	3: (* === Wait & process MB response *)
		IF NOT MB_Start THEN
			IF MB_MASTER.MB_Error=0 THEN
				CASE VARS[VarCnt].FunCode OF
					1,2,3,4:
						IF VARS[VarCnt].Variable_Size=200 THEN
							COPY_32SWAP16(ADR(MB_Resp.Data), VARS[VarCnt].Variable);
						ELSIF VARS[VarCnt].Variable_Size>1 THEN
							MEMCPY(ADR(MB_Resp.Data), VARS[VarCnt].Variable, 2*VARS[VarCnt].Variable_Size);
						ELSE
							VARS[VarCnt].Variable^:=MB_Resp.Data[0];
						END_IF
				END_CASE
				MB_Lock:=FALSE;
				(* Signal error recovery *)
				IF VARS_Alarm=TRUE AND VarCnt=VarAlarm THEN
					LogEv(EL_Wrn,EO_MODBUS,ID,5,'');
					VARS_Alarm:=FALSE;
				END_IF
				(* Next var *)
				VarCnt:=VarCnt+1;
				VarSta:=2;
			ELSE
				IF VarRetry<3 THEN
					VarRetry:=VarRetry+1;
					MB_Start:=TRUE;
				ELSE
					MB_Lock:=FALSE;
					(* Signal error *)
					IF VARS_Alarm=FALSE THEN
						LogEv(EL_Wrn,EO_MODBUS,ID,3,INT_TO_STRING(MB_MASTER.MB_Error));
						VARS_Alarm:=TRUE;
						VarAlarm:=VarCnt-1;
					END_IF
					(* Next var *)
					VarCnt:=VarCnt+1;
					VarSta:=2;
				END_IF
			END_IF
		END_IF

ELSE
	VarSta:=0;
END_CASE
END_ACTION

(* POU Utils Functions/TONOF, ST *)
FUNCTION_BLOCK TONOF
VAR_INPUT
	IN		: BOOL;
	PT_ON	: TIME; (* time to pass, before OUT is set *)
	PT_OF	: TIME; (* time to pass, before OUT is reset *)
END_VAR
VAR_OUTPUT
	OUT		: BOOL;
END_VAR
VAR
	timer	: TON;
END_VAR
IF IN<>OUT THEN
	timer(IN:=TRUE,PT:=SEL(IN,PT_OF,PT_ON));
	IF timer.Q THEN OUT:=IN; END_IF
ELSE
	timer(IN:=FALSE);
END_IF
END_FUNCTION_BLOCK

(* POU Plant_Objects/obj_COMPRESSORE_OLD, ST *)
FUNCTION_BLOCK obj_COMPRESSORE_OLD
VAR CONSTANT

	TimeOutModBus: TON;

END_VAR
VAR_INPUT
	ID			:	BYTE;
	Address		:	BYTE;


	(* Modbus *)
	Refresh_Now	:	BOOL;			(* Richiesta di lettura stato macchina Immediata  *)
	retryErrMax	:	BYTE := 2;

	OnOff		: 	BOOL;

	IndirizzoDaScrivere: WORD;
	DatoDaScrivere: INT;
	ScriviDato: BOOL;
	ScriviCoil: BOOL;

	fWriteAttivazioneComandi:BOOL;


	RUN_REQ: BOOL;
	STOP_REQ:BOOL;
	AgggiornoStartStop: BOOL;

	CARICO_REQ: BOOL;
	RELEASE_REQ: BOOL;

	LocSelManAuto:BOOL;
	LocOFP:INT;
	LocONP:INT;


END_VAR
VAR_IN_OUT
	ModBus		:obj_MODBUS;
END_VAR
VAR_OUTPUT
	Run			:	BOOL;

	Status_Log	:	WORD;
	Status_Vis	:	DWORD;
END_VAR
VAR
	(* da diego per gestione stato stringa > 255*)
	temp :STRING(255);
	tempRaw		: ARRAY [0..MAX_SEND_TCP_CLIENT] OF BYTE;
	tempRawLen :DINT;
	longString:STRING(255);

	(* Timer manage switch on/off delay *)
	Delay		: 	TONOF;
	Warning		:	FLT_TAP := (TAP:=100);
	AllarmeCompressore_MB		:	FLT_TAP;
	WarningCompressore_MB		:	FLT_TAP;
	AllarmeCompressoreAttivo_MB		:	FLT_TAP;
	RientrAllarmeCompressore_MB		:	FLT_TAP;
	RientrWarningCompressore_MB		:	FLT_TAP;

	AllarmeAttivo: INT;


	state		:	INT;
	retry		:	BYTE;
	retryErr	:	BYTE;
	ReadTmr		:	TON := (PT:=T#5s);
	fModbusAlr:BOOL;

	Ctrl_Run: BOOL;


	VerificaFuctionCode: INT;
	VerificaNodoLetto: INT;
	ErroreComuModBus: BOOL;
	IndiceErrore: BYTE;

	MB_BitStato: ARRAY [0..1] OF BOOL;
	MB_RegistriLetti: ARRAY [0..1] OF INT;
	MB_RegistriHoldingLetti: ARRAY [0..400] OF INT;
	MB_BitStatoCoil: ARRAY [0..1] OF BOOL;



	AddressRead: BYTE;
	index: BYTE;
	indexErr: BYTE;

	x: INT;
	IndirizzoStart: INT;
	Stop: BOOL;
	start: BOOL;
	StatusControl: ARRAY [0..15] OF BOOL;



	TOFF_RitardoAllarme: TOF;
	TOFF_RitardoWarning: TOF;
	trig_RitardoWarning: F_TRIG;
	trig_Ritardoallarme: F_TRIG;
	CompressoreInAllarme: BOOL;
	AllarmeAttivoSuCompressore: INT;
	CompressoreInWarning: BOOL;
	WarningAttivoSuCompressore: INT;
END_VAR
(* Call ModBus state machine *)
Stm();

(* Check alarm	*)
CheckAlarm();

(* Seganalzione stato Compressore  *)
IF ErroreComuModBus OR AllarmeCompressoreAttivo_MB.IN THEN (* corretto da DB 27/07/2017, era AllarmeCompressore_MB*)
		Status_Log:=2; Status_Vis:=16#2020F0;
   ELSIF WarningCompressore_MB.in  THEN
		Status_Log:=1; Status_Vis:=16#20F0F0;
    ELSE
		Status_Log:=0;
		Status_Vis:=16#006000;
END_IF
END_FUNCTION_BLOCK
ACTION AddLogData:
Logger.s1:=INSERT('&COMPINGRML=',BYTE_TO_STRING(ID),11);
IF ID<10 THEN Logger.s1:=INSERT(Logger.s1,'0',11); END_IF

FOR tempRawLen:=0 TO MAX_SEND_TCP_CLIENT DO
                tempRaw[tempRawLen]:=0;
END_FOR

tempRawLen:=0;


temp:=Logger.s1;
ADDSTRING(ADR(tempRaw), ADR(temp), tempRawLen);



temp:=CONCAT(WORD_TO_STRING(Status_Log),';');
ADDSTRING(ADR(tempRaw), ADR(temp), tempRawLen);


(* Sparo gli ingressi Digitali **)
FOR x:= 0 TO 15 DO
	temp:=CONCAT(SEL(StatusControl[x],'0','1'),';');
	ADDSTRING(ADR(tempRaw), ADR(temp), tempRawLen);
END_FOR

(*

temp:=CONCAT(INT_TO_STRING(MB_RegistriHoldingLetti[1]),';');
ADDSTRING(ADR(tempRaw), ADR(temp), tempRawLen);
temp:=CONCAT(INT_TO_STRING(MB_RegistriHoldingLetti[1]),';');
ADDSTRING(ADR(tempRaw), ADR(temp), tempRawLen); *)
temp:=CONCAT(INT_TO_STRING(MB_RegistriHoldingLetti[3]),';');
ADDSTRING(ADR(tempRaw), ADR(temp), tempRawLen);
temp:=CONCAT(INT_TO_STRING(MB_RegistriHoldingLetti[4]),';');
ADDSTRING(ADR(tempRaw), ADR(temp), tempRawLen);
temp:=CONCAT(INT_TO_STRING(MB_RegistriHoldingLetti[5]),';');
ADDSTRING(ADR(tempRaw), ADR(temp), tempRawLen);
temp:=CONCAT(INT_TO_STRING(MB_RegistriHoldingLetti[6]),';');
ADDSTRING(ADR(tempRaw), ADR(temp), tempRawLen);
temp:=CONCAT(INT_TO_STRING(MB_RegistriHoldingLetti[7]),';');
ADDSTRING(ADR(tempRaw), ADR(temp), tempRawLen);
temp:=CONCAT(INT_TO_STRING(MB_RegistriHoldingLetti[8]),';');
ADDSTRING(ADR(tempRaw), ADR(temp), tempRawLen);
temp:=CONCAT(INT_TO_STRING(MB_RegistriHoldingLetti[9]),';');
ADDSTRING(ADR(tempRaw), ADR(temp), tempRawLen);
temp:=CONCAT(INT_TO_STRING(MB_RegistriHoldingLetti[10]),';');
ADDSTRING(ADR(tempRaw), ADR(temp), tempRawLen);
temp:=CONCAT(INT_TO_STRING(MB_RegistriHoldingLetti[20]),';');
ADDSTRING(ADR(tempRaw), ADR(temp), tempRawLen);
temp:=CONCAT(INT_TO_STRING(MB_RegistriHoldingLetti[64]),';');
ADDSTRING(ADR(tempRaw), ADR(temp), tempRawLen);
temp:=CONCAT(INT_TO_STRING(MB_RegistriHoldingLetti[65]),';');
ADDSTRING(ADR(tempRaw), ADR(temp), tempRawLen);
temp:=CONCAT(INT_TO_STRING(MB_RegistriHoldingLetti[66]),';');
ADDSTRING(ADR(tempRaw), ADR(temp), tempRawLen);
temp:=CONCAT(INT_TO_STRING(MB_RegistriHoldingLetti[67]),';');
ADDSTRING(ADR(tempRaw), ADR(temp), tempRawLen);
temp:=CONCAT(INT_TO_STRING(MB_RegistriHoldingLetti[98]),';');
ADDSTRING(ADR(tempRaw), ADR(temp), tempRawLen);
temp:=CONCAT(INT_TO_STRING(MB_RegistriHoldingLetti[103]),';');
ADDSTRING(ADR(tempRaw), ADR(temp), tempRawLen);
temp:=CONCAT(INT_TO_STRING(MB_RegistriHoldingLetti[112]),';');
ADDSTRING(ADR(tempRaw), ADR(temp), tempRawLen);
temp:=CONCAT(INT_TO_STRING(MB_RegistriHoldingLetti[113]),';');
ADDSTRING(ADR(tempRaw), ADR(temp), tempRawLen);
temp:=CONCAT(INT_TO_STRING(MB_RegistriHoldingLetti[114]),';');
ADDSTRING(ADR(tempRaw), ADR(temp), tempRawLen);
temp:=CONCAT(INT_TO_STRING(MB_RegistriHoldingLetti[116]),';');
ADDSTRING(ADR(tempRaw), ADR(temp), tempRawLen);
temp:=CONCAT(INT_TO_STRING(MB_RegistriHoldingLetti[117]),';');
ADDSTRING(ADR(tempRaw), ADR(temp), tempRawLen);
temp:=CONCAT(INT_TO_STRING(MB_RegistriHoldingLetti[123]),';');
ADDSTRING(ADR(tempRaw), ADR(temp), tempRawLen);
temp:=CONCAT(INT_TO_STRING(MB_RegistriHoldingLetti[125]),';');
ADDSTRING(ADR(tempRaw), ADR(temp), tempRawLen);
temp:=CONCAT(INT_TO_STRING(MB_RegistriHoldingLetti[130]),';');
ADDSTRING(ADR(tempRaw), ADR(temp), tempRawLen);
temp:=CONCAT(INT_TO_STRING(MB_RegistriHoldingLetti[255]),';');
ADDSTRING(ADR(tempRaw), ADR(temp), tempRawLen);
temp:=CONCAT(INT_TO_STRING(MB_RegistriHoldingLetti[256]),';');
ADDSTRING(ADR(tempRaw), ADR(temp), tempRawLen);
temp:=CONCAT(INT_TO_STRING(MB_RegistriHoldingLetti[257]),';');
ADDSTRING(ADR(tempRaw), ADR(temp), tempRawLen);
temp:=CONCAT(INT_TO_STRING(MB_RegistriHoldingLetti[258]),';');
ADDSTRING(ADR(tempRaw), ADR(temp), tempRawLen);
temp:=CONCAT(INT_TO_STRING(MB_RegistriHoldingLetti[259]),';');
ADDSTRING(ADR(tempRaw), ADR(temp), tempRawLen);
temp:=CONCAT(INT_TO_STRING(MB_RegistriHoldingLetti[260]),';');
ADDSTRING(ADR(tempRaw), ADR(temp), tempRawLen);
temp:=CONCAT(INT_TO_STRING(MB_RegistriHoldingLetti[261]),';');
ADDSTRING(ADR(tempRaw), ADR(temp), tempRawLen);
temp:=CONCAT(INT_TO_STRING(MB_RegistriHoldingLetti[261]),';');
ADDSTRING(ADR(tempRaw), ADR(temp), tempRawLen);
temp:=CONCAT(INT_TO_STRING(MB_RegistriHoldingLetti[263]),';');
ADDSTRING(ADR(tempRaw), ADR(temp), tempRawLen);
temp:=CONCAT(INT_TO_STRING(MB_RegistriHoldingLetti[264]),';');
ADDSTRING(ADR(tempRaw), ADR(temp), tempRawLen);
temp:=CONCAT(INT_TO_STRING(MB_RegistriHoldingLetti[265]),';');
ADDSTRING(ADR(tempRaw), ADR(temp), tempRawLen);
temp:=CONCAT(INT_TO_STRING(MB_RegistriHoldingLetti[266]),';');
ADDSTRING(ADR(tempRaw), ADR(temp), tempRawLen);
temp:=CONCAT(INT_TO_STRING(MB_RegistriHoldingLetti[267]),';');
ADDSTRING(ADR(tempRaw), ADR(temp), tempRawLen);
temp:=CONCAT(INT_TO_STRING(MB_RegistriHoldingLetti[268]),';');
ADDSTRING(ADR(tempRaw), ADR(temp), tempRawLen);
temp:=CONCAT(INT_TO_STRING(MB_RegistriHoldingLetti[269]),';');
ADDSTRING(ADR(tempRaw), ADR(temp), tempRawLen);
temp:=(INT_TO_STRING(MB_RegistriHoldingLetti[270]));
ADDSTRING(ADR(tempRaw), ADR(temp), tempRawLen);


ADDSTRING(ADR(Logger.TData), ADR(tempRaw), Logger.TLen);
END_ACTION
ACTION CheckAlarm:
(**** GEstione Log ad Evento *****)



	AllarmeCompressoreAttivo_MB(IN:=CompressoreInAllarme AND AllarmeAttivoSuCompressore<>AllarmeAttivo );

	IF  AllarmeCompressoreAttivo_MB.EVH THEN
		LogEv(EL_Alarm,EO_COMPINGRML,ID,1,CONCAT ('AllarmeAttivo_n.', INT_TO_STRING(MB_RegistriHoldingLetti[256])));
		AllarmeAttivo:=MB_RegistriHoldingLetti[256];
	END_IF


	TOFF_RitardoAllarme(in:=CompressoreInAllarme,pt:=t#10s);    (* AllarmeAttivoSuCompressore=0 *)
	RientrAllarmeCompressore_MB(IN:=(TOFF_RitardoAllarme.Q) );

	IF  RientrAllarmeCompressore_MB.EVL  THEN
		LogEv(EL_Log,EO_COMPINGRML,ID,2,CONCAT ('AllarmeRientrato_n.', INT_TO_STRING(MB_RegistriHoldingLetti[256])));
		AllarmeAttivo:=0;
		AllarmeAttivoSuCompressore:=0;
	END_IF



	WarningCompressore_MB(IN:=CompressoreInWarning );

	IF WarningCompressore_MB.EVH THEN
		LogEv(EL_Wrn,EO_COMPINGRML,ID,1,CONCAT ('WarninigAttivo_n.', INT_TO_STRING(MB_RegistriHoldingLetti[255])));
	END_IF

	TOFF_RitardoWarning(in:=CompressoreInWarning,pt:=t#10s);   (* WarningAttivoSuCompressore=0*)
	RientrWarningCompressore_MB(IN:=(TOFF_RitardoWarning.Q) );

	IF RientrWarningCompressore_MB.EVL THEN
		LogEv(EL_Log,EO_COMPINGRML,ID,2,CONCAT ('WarningRientrato_n.', INT_TO_STRING(MB_RegistriHoldingLetti[255])));
	END_IF
END_ACTION
ACTION Stm:
CASE state OF
	0:	(* Refresh time manager *)
		ReadTmr(IN:=NOT ReadTmr.Q);
		(*A tempo interrogo il nodo sempre che non ci sia qualcuno che lo sta interrogando in quel momento *)

		IF (ReadTmr.Q AND NodoDaInterrogareCompressoreVecchio=Address )  AND NOT InibiscoModbusCompressoreVecchio THEN
			state := 10;
			ReadTmr.PT := T#100ms;  (* moreno *)
			Refresh_Now := FALSE;
			InibiscoModbusCompressoreVecchio := TRUE;
		END_IF

	(**** Leggo le Analogiche a Disposzione  ****)

	10:	(* richiedo lettura Holding Registere   *)

		Modbus.MB_Query.SlaveAddress := Address;
		Modbus.MB_Query.FunctionCode := 3;
		IndirizzoStart:=1;
		ModBus.MB_Query.Read_StartAddress :=IndirizzoStart - 1 ;
		ModBus.MB_Query.Read_Quantity := 2;
		ModBus.MB_Start := TRUE;
		state := 20;

	20:	(* Risposta all'interrogazione *)
		IF NOT ModBus.MB_Start   THEN
			VerificaFuctionCode:=ModBus.MB_Resp.FunctionCode;
			VerificaNodoLetto:=ModBus.MB_Resp.SlaveAddress;

			IF ModBus.MB_MASTER.MB_Error<>0 THEN
				state := 300;
			ELSE
				FOR x:=0 TO ModBus.MB_Query.Read_Quantity DO
					IF x+IndirizzoStart=3 THEN
						IF  ModBus.MB_Resp.Data[x]<260 THEN    (* condizione perchè questo registro si sporca con un valore 599 *)
				       		MB_RegistriHoldingLetti[x+IndirizzoStart] := ModBus.MB_Resp.Data[x];   	(* Vedi tabella *)
						ELSE
				       		MB_RegistriHoldingLetti[x+IndirizzoStart] := MB_RegistriHoldingLetti[x+IndirizzoStart];   	(* Vedi tabella *)
						END_IF
					ELSE
				       	MB_RegistriHoldingLetti[x+IndirizzoStart] := ModBus.MB_Resp.Data[x];   	(* Vedi tabella *)
					END_IF
				END_FOR

					StatusControl[0]:= MB_RegistriHoldingLetti[IndirizzoStart].0;   	(* Vedi tabella *)
					StatusControl[1]:= MB_RegistriHoldingLetti[IndirizzoStart].1;   	(* Vedi tabella *)
					StatusControl[2]:= MB_RegistriHoldingLetti[IndirizzoStart].2;   	(* Vedi tabella *)
					StatusControl[3]:= MB_RegistriHoldingLetti[IndirizzoStart].3;   	(* Vedi tabella *)
					StatusControl[4]:= MB_RegistriHoldingLetti[IndirizzoStart].4;   	(* Vedi tabella *)
					StatusControl[5]:= MB_RegistriHoldingLetti[IndirizzoStart].5;   	(* Vedi tabella *)
					StatusControl[6]:= MB_RegistriHoldingLetti[IndirizzoStart].6;   	(* Vedi tabella *)
					StatusControl[7]:= MB_RegistriHoldingLetti[IndirizzoStart].7;   	(* Vedi tabella *)
					StatusControl[8]:= MB_RegistriHoldingLetti[IndirizzoStart].8;   	(* Vedi tabella *)
					StatusControl[9]:= MB_RegistriHoldingLetti[IndirizzoStart].9;   	(* Vedi tabella *)
					StatusControl[10]:= MB_RegistriHoldingLetti[IndirizzoStart].10;   	(* Vedi tabella *)
					StatusControl[11]:= MB_RegistriHoldingLetti[IndirizzoStart].11;   	(* Vedi tabella *)
					StatusControl[12]:= MB_RegistriHoldingLetti[IndirizzoStart].12;   	(* Vedi tabella *)
					StatusControl[13]:= MB_RegistriHoldingLetti[IndirizzoStart].13;   	(* Vedi tabella *)
					StatusControl[14]:= MB_RegistriHoldingLetti[IndirizzoStart].14;   	(* Vedi tabella *)
					StatusControl[15]:= MB_RegistriHoldingLetti[IndirizzoStart].15;   	(* Vedi tabella *)


					CompressoreInAllarme:=StatusControl[6];
					CompressoreInWarning:=StatusControl[7];



				IndirizzoStart:=3;
				ModBus.MB_Query.Read_StartAddress :=IndirizzoStart-1; 	(* richiedo lettura altri Parametri *)
				ModBus.MB_Query.Read_Quantity := 19;
				ModBus.MB_Start := TRUE;

				state := 40;
			END_IF
		END_IF

	30: (* Rispota Altri paramenti *)
		IF NOT ModBus.MB_Start  THEN

			IF ModBus.MB_MASTER.MB_Error<>0 THEN
				state := 300;
			ELSE

				FOR x:=0 TO ModBus.MB_Query.Read_Quantity DO
					MB_RegistriHoldingLetti[x+IndirizzoStart] := ModBus.MB_Resp.Data[x];   	(* Vedi tabella *)
				END_FOR

				IndirizzoStart:=20;
				ModBus.MB_Query.Read_StartAddress :=IndirizzoStart-1; 	(* richiedo lettura altri Parametri *)
				ModBus.MB_Query.Read_Quantity := 1;
				ModBus.MB_Start := TRUE;

				state := 40;
			END_IF
		END_IF

	40: (* Rispota Altri paramenti *)
		IF NOT ModBus.MB_Start  THEN

			IF ModBus.MB_MASTER.MB_Error<>0 THEN
				state := 300;
			ELSE

				FOR x:=0 TO ModBus.MB_Query.Read_Quantity DO
					MB_RegistriHoldingLetti[x+IndirizzoStart] := ModBus.MB_Resp.Data[x];   	(* Vedi tabella *)
				END_FOR

				IndirizzoStart:=64;
				ModBus.MB_Query.Read_StartAddress :=IndirizzoStart-1; 	(* richiedo lettura altri Parametri *)
				ModBus.MB_Query.Read_Quantity := 4;
				ModBus.MB_Start := TRUE;

				state := 45;
			END_IF
		END_IF

	45: (* Rispota Altri paramenti *)
		IF NOT ModBus.MB_Start  THEN

			IF ModBus.MB_MASTER.MB_Error<>0 THEN
				state := 300;
			ELSE
				FOR x:=0 TO ModBus.MB_Query.Read_Quantity DO
					MB_RegistriHoldingLetti[x+IndirizzoStart] := ModBus.MB_Resp.Data[x];   	(* Vedi tabella *)
				END_FOR

				IndirizzoStart:=96;
				ModBus.MB_Query.Read_StartAddress :=IndirizzoStart-1; 	(* richiedo lettura altri Parametri *)
				ModBus.MB_Query.Read_Quantity := 8;
				ModBus.MB_Start := TRUE;

				state := 50;
			END_IF
		END_IF


	50: (* Rispota Altri paramenti *)
		IF NOT ModBus.MB_Start  THEN

			IF ModBus.MB_MASTER.MB_Error<>0 THEN
				state := 300;
			ELSE
				FOR x:=0 TO ModBus.MB_Query.Read_Quantity DO
					MB_RegistriHoldingLetti[x+IndirizzoStart] := ModBus.MB_Resp.Data[x];   	(* Vedi tabella *)
				END_FOR

				IndirizzoStart:=112;
				ModBus.MB_Query.Read_StartAddress :=IndirizzoStart-1; 	(* richiedo lettura altri Parametri *)
				ModBus.MB_Query.Read_Quantity := 10;
				ModBus.MB_Start := TRUE;


				state := 51;
			END_IF
		END_IF


	51: (* Rispota Altri paramenti *)
		IF NOT ModBus.MB_Start  THEN

			IF ModBus.MB_MASTER.MB_Error<>0 THEN
				state := 300;
			ELSE
				FOR x:=0 TO ModBus.MB_Query.Read_Quantity DO
					MB_RegistriHoldingLetti[x+IndirizzoStart] := ModBus.MB_Resp.Data[x];   	(* Vedi tabella *)
				END_FOR

				IndirizzoStart:=256;
				ModBus.MB_Query.Read_StartAddress :=IndirizzoStart-1; 	(* richiedo lettura altri Parametri *)
				ModBus.MB_Query.Read_Quantity := 14;
				ModBus.MB_Start := TRUE;


				state := 55;
			END_IF
		END_IF


	55: (* Rispota Altri paramenti *)
		IF NOT ModBus.MB_Start  THEN

			IF ModBus.MB_MASTER.MB_Error<>0 THEN
				state := 300;
			ELSE
				FOR x:=0 TO ModBus.MB_Query.Read_Quantity DO
					MB_RegistriHoldingLetti[x+IndirizzoStart] := ModBus.MB_Resp.Data[x];   	(* Vedi tabella *)
				END_FOR

				WarningAttivoSuCompressore:=MB_RegistriHoldingLetti[255];
				AllarmeAttivoSuCompressore:=MB_RegistriHoldingLetti[256];


				IndirizzoStart:=122;
				ModBus.MB_Query.Read_StartAddress :=IndirizzoStart-1; 	(* richiedo lettura altri Parametri *)
				ModBus.MB_Query.Read_Quantity := 10;
				ModBus.MB_Start := TRUE;

				state := 56;
			END_IF
		END_IF

	56: (* Rispota Altri paramenti *)
		IF NOT ModBus.MB_Start  THEN

			IF ModBus.MB_MASTER.MB_Error<>0 THEN
				state := 300;
			ELSE
				FOR x:=0 TO ModBus.MB_Query.Read_Quantity DO
					MB_RegistriHoldingLetti[x+IndirizzoStart] := ModBus.MB_Resp.Data[x];   	(* Vedi tabella *)
				END_FOR

				IndirizzoStart:=132;
				ModBus.MB_Query.Read_StartAddress :=IndirizzoStart-1; 	(* richiedo lettura altri Parametri *)
				ModBus.MB_Query.Read_Quantity := 10;
				ModBus.MB_Start := TRUE;

				state := 57;
			END_IF
		END_IF

	57: (* Rispota Altri paramenti *)
		IF NOT ModBus.MB_Start  THEN

			IF ModBus.MB_MASTER.MB_Error<>0 THEN
				state := 300;
			ELSE
				FOR x:=0 TO ModBus.MB_Query.Read_Quantity DO
					MB_RegistriHoldingLetti[x+IndirizzoStart] := ModBus.MB_Resp.Data[x];   	(* Vedi tabella *)
				END_FOR

				IndirizzoStart:=142;
				ModBus.MB_Query.Read_StartAddress :=IndirizzoStart-1; 	(* richiedo lettura altri Parametri *)
				ModBus.MB_Query.Read_Quantity := 10;
				ModBus.MB_Start := TRUE;

				state := 58;
			END_IF
		END_IF

	58: (* Rispota Altri paramenti *)
		IF NOT ModBus.MB_Start  THEN

			IF ModBus.MB_MASTER.MB_Error<>0 THEN
				state := 300;
			ELSE
				FOR x:=0 TO ModBus.MB_Query.Read_Quantity DO
					MB_RegistriHoldingLetti[x+IndirizzoStart] := ModBus.MB_Resp.Data[x];   	(* Vedi tabella *)
				END_FOR

				IndirizzoStart:=250;
				ModBus.MB_Query.Read_StartAddress :=IndirizzoStart-1; 	(* richiedo lettura altri Parametri *)
				ModBus.MB_Query.Read_Quantity := 6;
				ModBus.MB_Start := TRUE;

				state := 60;
			END_IF
		END_IF




	60: (* Rispota Altri paramenti *)
		IF NOT ModBus.MB_Start  THEN

			IF ModBus.MB_MASTER.MB_Error<>0 THEN
				state := 300;
			ELSE
				FOR x:=0 TO ModBus.MB_Query.Read_Quantity DO
					MB_RegistriHoldingLetti[x+IndirizzoStart] := ModBus.MB_Resp.Data[x];   	(* Vedi tabella *)
				END_FOR

				state :=290;
			END_IF
		END_IF


		290:    (* Scrittura il comando di run o stop da remoto*)
		IF NOT ModBus.MB_Start THEN
			IF ModBus.MB_MASTER.MB_Error<>0 THEN (*OR ModBus.MB_MASTER.MB_Error<>0 THEN*)
				state := 300;
			ELSE
				IF AgggiornoStartStop  THEN

					Modbus.MB_Query.FunctionCode := 6;
					Modbus.MB_Query.SlaveAddress := Address;

					IF RUN_REQ THEN
							IndirizzoDaScrivere:=1;
								 DatoDaScrivere:=MB_RegistriHoldingLetti[IndirizzoDaScrivere];
	  							 DatoDaScrivere.0:=TRUE;
  							        DatoDaScrivere.1:=TRUE;
							        DatoDaScrivere.2:=FALSE;
								 RUN_REQ:=FALSE;
					END_IF
					IF STOP_REQ THEN
							IndirizzoDaScrivere:=1;
								 DatoDaScrivere:=MB_RegistriHoldingLetti[IndirizzoDaScrivere];
	  							 DatoDaScrivere.0:=TRUE;
  							        DatoDaScrivere.1:=FALSE;
							        DatoDaScrivere.2:=FALSE;
								STOP_REQ:=FALSE;
					END_IF
					IF RELEASE_REQ THEN
							IndirizzoDaScrivere:=1;
								 DatoDaScrivere:=MB_RegistriHoldingLetti[IndirizzoDaScrivere];
	  							 DatoDaScrivere.0:=FALSE;
  							        DatoDaScrivere.1:=FALSE;
							        DatoDaScrivere.2:=FALSE;
								 RELEASE_REQ:=FALSE;
					END_IF
					IF CARICO_REQ THEN
							IndirizzoDaScrivere:=1;
								 DatoDaScrivere:=MB_RegistriHoldingLetti[IndirizzoDaScrivere];
	  							 DatoDaScrivere.0:=FALSE;
  							        DatoDaScrivere.1:=FALSE;
							        DatoDaScrivere.2:=TRUE;
								 CARICO_REQ:=FALSE;
					END_IF


					ModBus.MB_Query.Write_StartAddress := IndirizzoDaScrivere-1;
					ModBus.MB_Query.Write_Data[0] := DatoDaScrivere;
					ModBus.MB_Start := TRUE;


					AgggiornoStartStop:=FALSE;



					state := 291;
					ELSE
					state := 291;
				END_IF
			END_IF
		END_IF

		291:    (* Scrittura BOOL - COIL o WORD *)
		IF NOT ModBus.MB_Start THEN
			IF ModBus.MB_MASTER.MB_Error<>0 THEN (*OR ModBus.MB_MASTER.MB_Error<>0 THEN*)
				state := 300;
			ELSE
				IF LocSelManAuto THEN
					Modbus.MB_Query.FunctionCode := 6;
					Modbus.MB_Query.SlaveAddress := Address;
					ModBus.MB_Query.Write_StartAddress := 112-1;
					ModBus.MB_Query.Write_Quantity :=1;
					ModBus.MB_Query.Write_Data[0] := LocOFP;
					ModBus.MB_Start := TRUE;
					state := 292;
				ELSE
					state := 292;
				END_IF
			END_IF
		END_IF

		292:    (* Scrittura BOOL - COIL o WORD *)
		IF NOT ModBus.MB_Start THEN
			IF ModBus.MB_MASTER.MB_Error<>0 THEN (*OR ModBus.MB_MASTER.MB_Error<>0 THEN*)
				state := 300;
			ELSE
				IF LocSelManAuto THEN
					Modbus.MB_Query.FunctionCode := 6;
					Modbus.MB_Query.SlaveAddress := Address;
					ModBus.MB_Query.Write_StartAddress := 113-1;
					ModBus.MB_Query.Write_Quantity :=1;
					ModBus.MB_Query.Write_Data[0] := LocONP;
					ModBus.MB_Start := TRUE;
					state := 295;
				ELSE
					state := 295;
				END_IF
			END_IF
		END_IF





		295:
		IF NOT ModBus.MB_Start THEN
			IF ModBus.MB_MASTER.MB_Error<>0 THEN (*OR ModBus.MB_MASTER.MB_Error<>0 THEN*)
				state := 300;
			ELSE
				IF fModbusAlr THEN fModbusAlr := FALSE; END_IF
				NodoDaInterrogareCompressoreVecchio:=Address+1;
				InibiscoModbusCompressoreVecchio:=FALSE;
				retryErr := 0;
				retry := 0;
				state := 0;
					IF fModbusAlr=FALSE AND ErroreComuModBus=TRUE THEN
						LogEv(EL_Log,EO_COMPINGRR,ID,62,'ComunicazioneModBus_OK');
						ErroreComuModBus := FALSE;
				(*	WarningCtr := SEL(WarningCtr=0, WarningCtr-1, 0); *)
					END_IF


			END_IF
		END_IF



	(**** CHECK MODBUS ERROR ****)
	300: 	(* Release MODBUS *)
			InibiscoModbusCompressoreVecchio:=FALSE;
			(* Retries *)
			retry:=retry+1;
			IF retry>3 THEN
				retry:=0;

				(* Verify if slave is dead *)
				IF retryErr < retryErrMaX THEN
					retryErr := retryErr + 1;
				ELSE
					fModbusAlr := TRUE;
					(* Verify ModBus error	*)

					IF fModbusAlr AND ErroreComuModBus=FALSE THEN
						LogEv(EL_Alarm,EO_COMPINGRR,ID,61,CONCAT('ErroreModbus_',INT_TO_STRING(ModBus.MB_MASTER.MB_Error)));
						ErroreComuModBus := TRUE;
					END_IF
				END_IF

				END_IF
			Refresh_Now := FALSE;
			NodoDaInterrogareCompressoreVecchio:=Address+1;
			state:=0;
END_CASE




(* Controllo Time Out Ciclo ModBus *)

TimeOutModBus(In:=state<>0,PT:=t#3s);
IF TimeOutModBus.Q THEN
	State:=0;
	Refresh_Now:=TRUE;  (* Rilancio la lettura del nodo *)
	IF MODBUS.MB_Lock=TRUE THEN MODBUS.MB_Lock:=FALSE;END_IF
	IF InibiscoModbusCompressoreVecchio=TRUE THEN InibiscoModbusCompressoreVecchio:=FALSE;END_IF
	NodoDaInterrogareCompressoreVecchio:=Address+1;

END_IF
END_ACTION

(* POU Plant_Objects/obj_ESSICATORE, ST *)
FUNCTION_BLOCK obj_ESSICATORE
VAR CONSTANT

	TimeOutModBus: TON;


END_VAR
VAR_INPUT
	ID			:	BYTE;
	Address		:	BYTE;


	(* Modbus *)
	Refresh_Now	:	BOOL;			(* Richiesta di lettura stato macchina Immediata  *)
	retryErrMax	:	BYTE := 2;

	OnOff		: 	BOOL;

	IndirizzoDaScrivere: WORD;
	DatoDaScrivere: INT;
	ScriviDato: BOOL;
	ScriviCoil: BOOL;

	fWriteAttivazioneComandi:BOOL;

	RUN_REQ: BOOL;
	STOP_REQ:BOOL;
	AgggiornoStartStop: BOOL;
END_VAR
VAR_IN_OUT
	ModBus		:obj_MODBUS;
END_VAR
VAR_OUTPUT
	Run			:	BOOL;

	Status_Log	:	WORD;
	Status_Vis	:	DWORD;
END_VAR
VAR
	(* da diego per gestione stato stringa > 255*)
	temp :STRING(255);
	tempRaw		: ARRAY [0..MAX_SEND_TCP_CLIENT] OF BYTE;
	tempRawLen :DINT;
	longString:STRING(255);

	(* Timer manage switch on/off delay *)
	Delay		: 	TONOF;
	Warning		:	FLT_TAP := (TAP:=100);
	AllarmeCompressore_MB		:	FLT_TAP;

	state		:	INT;
	retry		:	BYTE;
	retryErr	:	BYTE;
	ReadTmr		:	TON := (PT:=T#5s);
	fModbusAlr:BOOL;

	Ctrl_Run: BOOL;


	VerificaFuctionCode: INT;
	VerificaNodoLetto: INT;
	ErroreComuModBus: BOOL;
	IndiceErrore: BYTE;

	MB_BitStato: ARRAY [0..1] OF BOOL;
	MB_RegistriLetti: ARRAY [0..1] OF INT;
	MB_RegistriHoldingLetti: ARRAY [0..500] OF INT;
	MB_BitStatoCoil: ARRAY [0..1] OF BOOL;



	AddressRead: BYTE;
	index: BYTE;
	indexErr: BYTE;





	x: INT;
	moreno1: INT;
	moreno2: INT;
	IndirizzoStart: INT;

	Parametro1280: WORD;
	Parametro1282: WORD;
	morenoind: INT;
	morenoqta: INT;
	Probe1: INT;
	StatusProbe1: INT;
	Probe2: INT;
	StatusProbe2: INT;
	Probe3: INT;
	StatusProbe3: INT;
	Probe4: INT;
	StatusProbe4: INT;
	TempoPausa: TON;
	IndirizzoTest: INT;
	FunctionTest: BYTE := 3;
	StatusMachine: BOOL;
	ChillerSet: INT;
	HoursWorking: WORD;
	SpeedCompressor: INT:=9999;
	faultEssicatore: BOOL;
	test: INT;
	Morenotest: WORD;
	Morenotest1: INT;
END_VAR
(* Call ModBus state machine *)
Stm();

(* Check alarm	*)

(* Seganalzione stato Compressore  *)
IF ErroreComuModBus THEN
		Status_Log:=2; Status_Vis:=16#2020F0;
(*	ELSIF Warning OR Warning2 THEN
		Status_Log:=1; Status_Vis:=16#20F0F0; *)
    ELSE
		Status_Log:=0;
		Status_Vis:=16#006000;
END_IF
END_FUNCTION_BLOCK
ACTION AddLogData:
Logger.s1:=CONCAT('&','ESC');
IF ID<10 THEN Logger.s1:=CONCAT(Logger.s1,'0');END_IF
Logger.s1:=CONCAT(Logger.s1,BYTE_TO_STRING(ID));
Logger.s1:=CONCAT(Logger.s1,'=');


FOR tempRawLen:=0 TO MAX_SEND_TCP_CLIENT DO
                tempRaw[tempRawLen]:=0;
END_FOR

tempRawLen:=0;


temp:=Logger.s1;
ADDSTRING(ADR(tempRaw), ADR(temp), tempRawLen);

temp:=CONCAT(WORD_TO_STRING(Status_Log),';');
ADDSTRING(ADR(tempRaw), ADR(temp), tempRawLen);

temp:=CONCAT(INT_TO_STRING(Probe1),';');
ADDSTRING(ADR(tempRaw), ADR(temp), tempRawLen);

temp:=CONCAT(BOOL_TO_STRING(StatusMachine),';');
ADDSTRING(ADR(tempRaw), ADR(temp), tempRawLen);

temp:=CONCAT(INT_TO_STRING(ChillerSet),';');
ADDSTRING(ADR(tempRaw), ADR(temp), tempRawLen);

temp:=CONCAT(INT_TO_STRING(HoursWorking),';');
ADDSTRING(ADR(tempRaw), ADR(temp), tempRawLen);

temp:=(INT_TO_STRING(SpeedCompressor));
ADDSTRING(ADR(tempRaw), ADR(temp), tempRawLen);


ADDSTRING(ADR(Logger.TData), ADR(tempRaw), Logger.TLen);
END_ACTION
ACTION Stm:
CASE state OF
	0:	(* Refresh time manager *)
		ReadTmr(IN:=NOT ReadTmr.Q);
		(*A tempo interrogo il nodo sempre che non ci sia qualcuno che lo sta interrogando in quel momento *)

		IF (ReadTmr.Q  ) OR Refresh_Now  THEN
			state := 10;
			ReadTmr.PT := T#500ms;  (* moreno *)
			Refresh_Now := FALSE;
			InibiscoModbusEssicatore := TRUE;
			TempoPausa(IN:=FALSE , PT:=t#200ms , Q=> , ET=> );

		END_IF

	(**** Leggo le Analogiche a Disposzione  ****)

	10:	(* richiedo lettura Holding Registere   *)


		Modbus.MB_MASTER.cbsCOM_BYTESIZE:=BS_8;
		Modbus.MB_MASTER.cpCOM_PARITY:=PARITY_NO;


		Modbus.MB_Query.SlaveAddress := Address;
		Modbus.MB_Query.FunctionCode := 3; (*3; *)
		IndirizzoStart:=257; (*257; *)
		ModBus.MB_Query.Read_StartAddress :=IndirizzoStart-1  ;
		ModBus.MB_Query.Read_Quantity := 2;(*19;*)
		ModBus.MB_Start := TRUE;

		state := 17;

	17: TempoPausa(IN:=TRUE , PT:=t#500ms , Q=> , ET=> );
			IF TempoPausa.Q THEN
			ModBus.MB_Start := TRUE;
			TempoPausa(IN:=FALSE , PT:=t#200ms , Q=> , ET=> );
				state := state+1;;
			END_IF
	18:	(* Risposta all'interrogazione *)
		IF NOT ModBus.MB_Start   THEN
			VerificaFuctionCode:=ModBus.MB_Resp.FunctionCode;
			VerificaNodoLetto:=ModBus.MB_Resp.SlaveAddress;

			IF ModBus.MB_MASTER.MB_Error=0 THEN
				Probe1:=ModBus.MB_Resp.Data[0];
				StatusProbe1:=ModBus.MB_Resp.Data[1];
			END_IF
				IndirizzoStart:=259;
				ModBus.MB_Query.Read_StartAddress :=IndirizzoStart - 1 ;
				ModBus.MB_Query.Read_Quantity :=2;
				state :=19;
			END_IF

	19: TempoPausa(IN:=TRUE , PT:=t#500ms , Q=> , ET=> );
			IF TempoPausa.Q THEN
			ModBus.MB_Start := TRUE;
			TempoPausa(IN:=FALSE , PT:=t#200ms , Q=> , ET=> );
				state := state+1;;
			END_IF

	20:	(* Risposta all'interrogazione *)
		IF NOT ModBus.MB_Start   THEN
			VerificaFuctionCode:=ModBus.MB_Resp.FunctionCode;
			VerificaNodoLetto:=ModBus.MB_Resp.SlaveAddress;

			IF ModBus.MB_MASTER.MB_Error=0 THEN
				Probe2:=ModBus.MB_Resp.Data[0];
				StatusProbe2:=ModBus.MB_Resp.Data[1];
			END_IF

				IndirizzoStart:=261;
				ModBus.MB_Query.Read_StartAddress :=IndirizzoStart - 1 ;
				ModBus.MB_Query.Read_Quantity :=2;

				state := 29;
		END_IF
	29: TempoPausa(IN:=TRUE , PT:=t#500ms , Q=> , ET=> );
			IF TempoPausa.Q THEN
				ModBus.MB_Start := TRUE;
				TempoPausa(IN:=FALSE , PT:=t#200ms , Q=> , ET=> );
				state := state+1;;
			END_IF
	30: (* Rispota Altri paramenti *)
		IF NOT ModBus.MB_Start  THEN

			IF ModBus.MB_MASTER.MB_Error=0 THEN
				Probe3:=ModBus.MB_Resp.Data[0];
				StatusProbe3:=ModBus.MB_Resp.Data[1];
			END_IF



				IndirizzoStart:=263;
				ModBus.MB_Query.Read_StartAddress :=IndirizzoStart - 1 ;
				ModBus.MB_Query.Read_Quantity := 2;

				state := 34;
			END_IF

	34: TempoPausa(IN:=TRUE , PT:=t#500ms , Q=> , ET=> );
			IF TempoPausa.Q THEN
				ModBus.MB_Start := TRUE;
				TempoPausa(IN:=FALSE , PT:=t#200ms , Q=> , ET=> );
				state := state+1;;
			END_IF

	35: (* Rispota Altri paramenti *)
		IF NOT ModBus.MB_Start  THEN

			IF ModBus.MB_MASTER.MB_Error=0 THEN
				Probe4:=ModBus.MB_Resp.Data[0];
				StatusProbe4:=ModBus.MB_Resp.Data[1];
			END_IF

				IndirizzoStart:=1281;
				ModBus.MB_Query.Read_StartAddress :=IndirizzoStart - 1 ;
				ModBus.MB_Query.Read_Quantity := 2;

				state := 41;
		END_IF

	41: TempoPausa(IN:=TRUE , PT:=t#500ms , Q=> , ET=> );
			IF TempoPausa.Q THEN
				ModBus.MB_Start := TRUE;
				TempoPausa(IN:=FALSE , PT:=t#200ms , Q=> , ET=> );
				state := state+1;;
			END_IF
	42: (* Rispota Altri paramenti *)
		IF NOT ModBus.MB_Start  THEN

			IF ModBus.MB_MASTER.MB_Error=0 THEN

				StatusMachine:=(ModBus.MB_Resp.Data[0].0);

			END_IF

				IndirizzoStart:=1537;
				ModBus.MB_Query.Read_StartAddress :=IndirizzoStart - 1 ;
				ModBus.MB_Query.Read_Quantity := 1;

				state := 43;
		END_IF


	43: TempoPausa(IN:=TRUE , PT:=t#500ms , Q=> , ET=> );
			IF TempoPausa.Q THEN
				ModBus.MB_Start := TRUE;
				TempoPausa(IN:=FALSE , PT:=t#200ms , Q=> , ET=> );
				state := state+1;;
			END_IF
	44: (* Rispota Altri paramenti *)
		IF NOT ModBus.MB_Start  THEN

			IF ModBus.MB_MASTER.MB_Error=0 THEN

				ChillerSet:=(ModBus.MB_Resp.Data[0]);
			END_IF

				IndirizzoStart:=3585;
				ModBus.MB_Query.Read_StartAddress :=IndirizzoStart - 1 ;
				ModBus.MB_Query.Read_Quantity := 1;

				state := 45;
		END_IF

	45: TempoPausa(IN:=TRUE , PT:=t#500ms , Q=> , ET=> );
			IF TempoPausa.Q THEN
				ModBus.MB_Start := TRUE;
				TempoPausa(IN:=FALSE , PT:=t#200ms , Q=> , ET=> );
				state := state+1;;
			END_IF
	46: (* Rispota Altri paramenti *)
		IF NOT ModBus.MB_Start  THEN

			IF ModBus.MB_MASTER.MB_Error=0 THEN

				HoursWorking:=(ModBus.MB_Resp.Data[0]);



			END_IF

				IndirizzoStart:=2049;
				ModBus.MB_Query.Read_StartAddress :=IndirizzoStart - 1 ;
				ModBus.MB_Query.Read_Quantity := 2;

				state := 47;
		END_IF

	47: TempoPausa(IN:=TRUE , PT:=t#500ms , Q=> , ET=> );
			IF TempoPausa.Q THEN
				ModBus.MB_Start := TRUE;
				TempoPausa(IN:=FALSE , PT:=t#200ms , Q=> , ET=> );
				state := state+1;;
			END_IF
	48: (* Rispota Altri paramenti *)
		IF NOT ModBus.MB_Start  THEN

			IF ModBus.MB_MASTER.MB_Error=0 THEN

				faultEssicatore:=(ModBus.MB_Resp.Data[0].3);
				Morenotest:=ModBus.MB_Resp.Data[0];
				Morenotest1:=ModBus.MB_Resp.Data[1];
			END_IF

				state := 295;
		END_IF


		295:
		IF NOT ModBus.MB_Start THEN
			IF ModBus.MB_MASTER.MB_Error<>0 THEN (*OR ModBus.MB_MASTER.MB_Error<>0 THEN*)
				state := 300;
			ELSE
				IF fModbusAlr THEN fModbusAlr := FALSE; END_IF
				NodoDaInterrogareEssicatore:=Address+1;
				InibiscoModbusEssicatore:=FALSE;
				retryErr := 0;
				retry := 0;
				state := 0;
					IF fModbusAlr=FALSE AND ErroreComuModBus=TRUE THEN
						LogEv(EL_Log,EO_COMPINGRML,ID,62,'ComunicazioneModBus_OK');
						ErroreComuModBus := FALSE;
				(*	WarningCtr := SEL(WarningCtr=0, WarningCtr-1, 0); *)
					END_IF
			END_IF


		END_IF




	(**** CHECK MODBUS ERROR ****)
	300: 	(* Release MODBUS *)
			InibiscoModbusEssicatore:=FALSE;
			(* Retries *)
			retry:=retry+1;
			IF retry>3 THEN
				retry:=0;

				(* Verify if slave is dead *)
				IF retryErr < retryErrMaX THEN
					retryErr := retryErr + 1;
				ELSE
					fModbusAlr := TRUE;
					(* Verify ModBus error	*)

					IF fModbusAlr AND ErroreComuModBus=FALSE THEN
						LogEv(EL_Alarm,EO_COMPINGRML,ID,61,CONCAT('ErroreModbus_',INT_TO_STRING(ModBus.MB_MASTER.MB_Error)));
						ErroreComuModBus := TRUE;
					END_IF
				END_IF

				END_IF
			Refresh_Now := FALSE;
			NodoDaInterrogareEssicatore:=Address+1;
			state:=0;
END_CASE




(* Controllo Time Out Ciclo ModBus *)

TimeOutModBus(In:=state<>0,PT:=t#30s);
IF TimeOutModBus.Q THEN
	State:=0;
	IF MODBUS.MB_Lock=TRUE THEN MODBUS.MB_Lock:=FALSE;END_IF
	IF InibiscoModbusEssicatore=TRUE THEN InibiscoModbusEssicatore:=FALSE;END_IF
	NodoDaInterrogareEssicatore:=Address+1;

END_IF
END_ACTION

(* POU Plant_Objects/obj_ESSICATORE_NEW, ST *)
FUNCTION_BLOCK obj_ESSICATORE_NEW
VAR CONSTANT

	TimeOutModBus: TON;


END_VAR
VAR_INPUT
	ID			:	BYTE;
	Address		:	BYTE;


	(* Modbus *)
	Refresh_Now	:	BOOL;			(* Richiesta di lettura stato macchina Immediata  *)
	retryErrMax	:	BYTE := 2;

	OnOff		: 	BOOL;

	IndirizzoDaScrivere: WORD;
	DatoDaScrivere: INT;
	ScriviDato: BOOL;
	ScriviCoil: BOOL;

	fWriteAttivazioneComandi:BOOL;

	RUN_REQ: BOOL;
	STOP_REQ:BOOL;
	AgggiornoStartStop: BOOL;
END_VAR
VAR_IN_OUT
	ModBus		:obj_MODBUS_Free;
END_VAR
VAR_OUTPUT
	Run			:	BOOL;

	Status_Log	:	WORD;
	Status_Vis	:	DWORD;
END_VAR
VAR
	(* da diego per gestione stato stringa > 255*)
	temp :STRING(255);
	tempRaw		: ARRAY [0..MAX_SEND_TCP_CLIENT] OF BYTE;
	tempRawLen :DINT;
	longString:STRING(255);

	(* Timer manage switch on/off delay *)
	Delay		: 	TONOF;
	Warning		:	FLT_TAP := (TAP:=100);
	AllarmeCompressore_MB		:	FLT_TAP;

	state		:	INT;
	retry		:	BYTE;
	retryErr	:	BYTE;
	ReadTmr		:	TON := (PT:=T#5s);
	fModbusAlr:BOOL;

	Ctrl_Run: BOOL;


	VerificaFuctionCode: INT;
	VerificaNodoLetto: INT;
	ErroreComuModBus: BOOL;
	IndiceErrore: BYTE;

	MB_BitStato: ARRAY [0..1] OF BOOL;
	MB_RegistriLetti: ARRAY [0..1] OF INT;
	MB_RegistriHoldingLetti: ARRAY [0..500] OF INT;
	MB_BitStatoCoil: ARRAY [0..1] OF BOOL;



	AddressRead: BYTE;
	index: BYTE;
	indexErr: BYTE;





	x: INT;
	moreno1: INT;
	moreno2: INT;
	IndirizzoStart: INT;

	Parametro1280: WORD;
	Parametro1282: WORD;
	morenoind: INT;
	morenoqta: INT;
	Probe1: INT;
	StatusProbe1: INT;
	Probe2: INT;
	StatusProbe2: INT;
	Probe3: INT;
	StatusProbe3: INT;
	Probe4: INT;
	StatusProbe4: INT;
	TempoPausa: TON;
	qta: INT := 1;
	ind: INT := 1;
	Probe1_1: WORD;
	Probe2_1: WORD;
	test: BOOL;
	alarmstatus: INT;
	Servicestatus: INT;
	StatusMachine: INT;
	CompressorSpeed: INT;
	WorkingHours: INT;
	AllarmeAttivo: INT;
	ton_AllarmeAttivo: TON;
	AllarmeStrumento_MB			:	FLT_TAP;
	RietrAllarmeStrumento_MB		:	FLT_TAP;




	test1: INT;
	test2: INT;
	test3: INT;
	test4: INT;
	test5: INT;
END_VAR
(* Call ModBus state machine *)
Stm();

(* Check alarm	*)
CheckAlarm();




(* Seganalzione stato Compressore  *)
IF ErroreComuModBus  OR AllarmeAttivo<>0 THEN
		Status_Log:=2; Status_Vis:=16#2020F0;
(*	ELSIF Warning OR Warning2 THEN
		Status_Log:=1; Status_Vis:=16#20F0F0; *)
    ELSE
		Status_Log:=0;
		Status_Vis:=16#006000;
END_IF
END_FUNCTION_BLOCK
ACTION AddLogData:
Logger.s1:=CONCAT('&','ESC');
IF ID<10 THEN Logger.s1:=CONCAT(Logger.s1,'0');END_IF
Logger.s1:=CONCAT(Logger.s1,BYTE_TO_STRING(ID));
Logger.s1:=CONCAT(Logger.s1,'=');


FOR tempRawLen:=0 TO MAX_SEND_TCP_CLIENT DO
                tempRaw[tempRawLen]:=0;
END_FOR

tempRawLen:=0;


temp:=Logger.s1;
ADDSTRING(ADR(tempRaw), ADR(temp), tempRawLen);

temp:=CONCAT(WORD_TO_STRING(Status_Log),';');
ADDSTRING(ADR(tempRaw), ADR(temp), tempRawLen);

temp:=CONCAT(INT_TO_STRING(Probe1),';');
ADDSTRING(ADR(tempRaw), ADR(temp), tempRawLen);

temp:=CONCAT(BOOL_TO_STRING(StatusMachine.0),';');
ADDSTRING(ADR(tempRaw), ADR(temp), tempRawLen);

temp:=CONCAT(INT_TO_STRING(9999),';');
ADDSTRING(ADR(tempRaw), ADR(temp), tempRawLen);

temp:=CONCAT(INT_TO_STRING(WorkingHours),';');
ADDSTRING(ADR(tempRaw), ADR(temp), tempRawLen);

temp:=(INT_TO_STRING(CompressorSpeed));
ADDSTRING(ADR(tempRaw), ADR(temp), tempRawLen);


ADDSTRING(ADR(Logger.TData), ADR(tempRaw), Logger.TLen);
END_ACTION
ACTION CheckAlarm:
(**** GEstione Log ad Evento *****)





	ton_AllarmeAttivo(IN:=AllarmeAttivo<>Alarmstatus,PT:=t#2s);

	AllarmeStrumento_MB(IN:=ton_AllarmeAttivo.Q );
	IF AllarmeStrumento_MB.EVH THEN
		LogEv(EL_Alarm,EO_COMPINGRR,ID,1,CONCAT ('NuovoAllarmeAttivo_n.', INT_TO_STRING(Alarmstatus)));
		AllarmeAttivo:=Alarmstatus; (*AllarmeAttivosuCTB;*)
	END_IF

	RietrAllarmeStrumento_MB(IN:=Alarmstatus<>0);

	IF RietrAllarmeStrumento_MB.EVL THEN
		LogEv(EL_Log,EO_COMPINGRR,ID,2,CONCAT ('AllarmeRientrato_EventualeAllarme_n.', INT_TO_STRING(Alarmstatus)));
		AllarmeAttivo:=Alarmstatus;
	END_IF
END_ACTION
ACTION Stm:
CASE state OF
	0:	(* Refresh time manager *)
		ReadTmr(IN:=NOT ReadTmr.Q);
		(*A tempo interrogo il nodo sempre che non ci sia qualcuno che lo sta interrogando in quel momento *)

		IF (ReadTmr.Q  ) OR Refresh_Now  THEN
			state := 10;
			ReadTmr.PT := T#500ms;  (* moreno *)
			Refresh_Now := FALSE;
			InibiscoModbusEssicatore := TRUE;
			TempoPausa(IN:=FALSE , PT:=t#200ms , Q=> , ET=> );

		END_IF

	(**** Leggo le Analogiche a Disposzione  ****)

	10:	(* richiedo lettura Holding Registere   *)


		Modbus.MB_MASTER.cbsCOM_BYTESIZE:=BS_7;
		Modbus.MB_MASTER.cpCOM_PARITY:=PARITY_EVEN;
		Modbus.ASCIIMODE:=TRUE;

		Modbus.MB_Query.SlaveAddress := Address;
		Modbus.MB_Query.FunctionCode := 3;
		IndirizzoStart:=0;
		ModBus.MB_Query.Read_StartAddress :=IndirizzoStart  ;
		ModBus.MB_Query.Read_Quantity := 4;(*19;*)
		state := 17;

	17: TempoPausa(IN:=TRUE , PT:=t#100ms , Q=> , ET=> );
			IF TempoPausa.Q THEN
				ModBus.MB_Start := TRUE;
				TempoPausa(IN:=FALSE , PT:=t#200ms , Q=> , ET=> );
				state := state+1;;
			END_IF


	18:	(* Risposta all'interrogazione *)
		IF NOT ModBus.MB_Start   THEN
			VerificaFuctionCode:=ModBus.MB_Resp.FunctionCode;
			VerificaNodoLetto:=ModBus.MB_Resp.SlaveAddress;

			IF ModBus.MB_MASTER.MB_Error=0 THEN
			(*	test:=RTU_TO_ASCIIRTU_TO_ASCII(Count, SendBuffer)( *)
				Probe1:=ModBus.MB_Resp.Data[0];
				Probe2:=ModBus.MB_Resp.Data[1];
				Probe3:=ModBus.MB_Resp.Data[2];
				Probe4:=ModBus.MB_Resp.Data[3];
			END_IF

		IndirizzoStart:=103;
		ModBus.MB_Query.Read_StartAddress :=IndirizzoStart  ;
		ModBus.MB_Query.Read_Quantity := 4;(*19;*)
		state :=27; (* 27; *)
		END_IF
	27: TempoPausa(IN:=TRUE , PT:=t#100ms , Q=> , ET=> );
			IF TempoPausa.Q THEN
				ModBus.MB_Start := TRUE;
				TempoPausa(IN:=FALSE , PT:=t#200ms , Q=> , ET=> );
				state := state+1;;
			END_IF


	28:	(* Risposta all'interrogazione *)
		IF NOT ModBus.MB_Start   THEN
			VerificaFuctionCode:=ModBus.MB_Resp.FunctionCode;
			VerificaNodoLetto:=ModBus.MB_Resp.SlaveAddress;

			IF ModBus.MB_MASTER.MB_Error=0 THEN
			(*	test:=RTU_TO_ASCIIRTU_TO_ASCII(Count, SendBuffer)( *)
				test1:=ModBus.MB_Resp.Data[0];
				test2:=ModBus.MB_Resp.Data[1];
				test3:=ModBus.MB_Resp.Data[2];
				test4:=ModBus.MB_Resp.Data[3];

				StatusMachine:=test1;
				CompressorSpeed:=test4;
			END_IF
			IndirizzoStart:=113;
			ModBus.MB_Query.Read_StartAddress :=IndirizzoStart  ;
			ModBus.MB_Query.Read_Quantity := 5;(*19;*)


			state :=29;
		END_IF

	29: TempoPausa(IN:=TRUE , PT:=t#100ms , Q=> , ET=> );
			IF TempoPausa.Q THEN
				ModBus.MB_Start := TRUE;
				TempoPausa(IN:=FALSE , PT:=t#200ms , Q=> , ET=> );
				state := state+1;;
			END_IF


	30:	(* Risposta all'interrogazione *)
		IF NOT ModBus.MB_Start   THEN
			VerificaFuctionCode:=ModBus.MB_Resp.FunctionCode;
			VerificaNodoLetto:=ModBus.MB_Resp.SlaveAddress;

			IF ModBus.MB_MASTER.MB_Error=0 THEN
			(*	test:=RTU_TO_ASCIIRTU_TO_ASCII(Count, SendBuffer)( *)
				test1:=ModBus.MB_Resp.Data[0];
				test2:=ModBus.MB_Resp.Data[1];
				test3:=ModBus.MB_Resp.Data[2];
				test4:=ModBus.MB_Resp.Data[3];
				test5:=ModBus.MB_Resp.Data[4];

				WorkingHours:=test2;
				Alarmstatus:=test3;


			END_IF

			state :=295;
		END_IF











		290:    (* Scrittura il comando di run o stop da remoto*)
		IF NOT ModBus.MB_Start THEN
			IF ModBus.MB_MASTER.MB_Error<>0 THEN (*OR ModBus.MB_MASTER.MB_Error<>0 THEN*)
				state := 300;
			ELSE
				IF AgggiornoStartStop  THEN

					Modbus.MB_Query.FunctionCode := 6;
					Modbus.MB_Query.SlaveAddress := Address;
					ModBus.MB_Query.Write_StartAddress := IndirizzoDaScrivere;
					ModBus.MB_Query.Write_Quantity :=1;


					 DatoDaScrivere:=MB_RegistriHoldingLetti[IndirizzoDaScrivere];
	  				 DatoDaScrivere.0:=FALSE;

					IF RUN_REQ THEN
								 DatoDaScrivere:=MB_RegistriHoldingLetti[IndirizzoDaScrivere];
	  							 DatoDaScrivere.0:=TRUE;
  							        DatoDaScrivere.1:=TRUE;
					END_IF
					IF STOP_REQ THEN
								 DatoDaScrivere:=MB_RegistriHoldingLetti[IndirizzoDaScrivere];
	  							 DatoDaScrivere.0:=TRUE;
  							        DatoDaScrivere.1:=FALSE;
					END_IF


					ModBus.MB_Query.Write_Data[0] := DatoDaScrivere;
					ModBus.MB_Start := TRUE;
					state := 291;
					AgggiornoStartStop:=FALSE;
				ELSE
					state := 291;
				END_IF
			END_IF
		END_IF
		291:    (* Scrittura BOOL - COIL o WORD *)
		IF NOT ModBus.MB_Start THEN
			IF ModBus.MB_MASTER.MB_Error<>0 THEN (*OR ModBus.MB_MASTER.MB_Error<>0 THEN*)
				state := 300;
			ELSE
				IF ScriviDato THEN
					IF ScriviCoil THEN
						Modbus.MB_Query.FunctionCode := 5;
					ELSE
						Modbus.MB_Query.FunctionCode := 6;
					END_IF
					Modbus.MB_Query.SlaveAddress := Address;
					ModBus.MB_Query.Write_StartAddress := IndirizzoDaScrivere-1;
					ModBus.MB_Query.Write_Quantity :=1;
					ModBus.MB_Query.Write_Data[0] := DatoDaScrivere;
					ModBus.MB_Start := TRUE;
						IF ScriviCoil THEN
							IF 	MB_BitStato[IndirizzoDaScrivere]=WORD_TO_BOOL(DatoDaScrivere-1) THEN
								ScriviDato:=FALSE;
							END_IF
						ELSE
							IF 	MB_RegistriHoldingLetti[IndirizzoDaScrivere]=DatoDaScrivere THEN
								ScriviDato:=FALSE;
							END_IF
						END_IF
					state := 295;
				ELSE
					state := 295;
				END_IF
			END_IF
		END_IF




		295:
		IF NOT ModBus.MB_Start THEN
			IF ModBus.MB_MASTER.MB_Error<>0 THEN (*OR ModBus.MB_MASTER.MB_Error<>0 THEN*)
				state := 300;
			ELSE
				IF fModbusAlr THEN fModbusAlr := FALSE; END_IF
				NodoDaInterrogareEssicatore:=Address+1;
				InibiscoModbusEssicatore:=FALSE;
				retryErr := 0;
				retry := 0;
				state := 0;
					IF fModbusAlr=FALSE AND ErroreComuModBus=TRUE THEN
						LogEv(EL_Log,EO_COMPINGRML,ID,62,'ComunicazioneModBus_OK');
						ErroreComuModBus := FALSE;
				(*	WarningCtr := SEL(WarningCtr=0, WarningCtr-1, 0); *)
					END_IF
			END_IF


		END_IF




	(**** CHECK MODBUS ERROR ****)
	300: 	(* Release MODBUS *)
			InibiscoModbusEssicatore:=FALSE;
			(* Retries *)
			retry:=retry+1;
			IF retry>3 THEN
				retry:=0;

				(* Verify if slave is dead *)
				IF retryErr < retryErrMaX THEN
					retryErr := retryErr + 1;
				ELSE
					fModbusAlr := TRUE;
					(* Verify ModBus error	*)

					IF fModbusAlr AND ErroreComuModBus=FALSE THEN
						LogEv(EL_Alarm,EO_COMPINGRML,ID,61,CONCAT('ErroreModbus_',INT_TO_STRING(ModBus.MB_MASTER.MB_Error)));
						ErroreComuModBus := TRUE;
					END_IF
				END_IF

				END_IF
			Refresh_Now := FALSE;
			NodoDaInterrogareEssicatore:=Address+1;
			state:=0;
END_CASE




(* Controllo Time Out Ciclo ModBus *)

TimeOutModBus(In:=state<>0,PT:=t#10s);
IF TimeOutModBus.Q THEN
	State:=0;
	ModBus.MB_Start := FALSE;

	(*Refresh_Now:=TRUE;  (* Rilancio la lettura del nodo *) *)
	IF MODBUS.MB_Lock=TRUE THEN MODBUS.MB_Lock:=FALSE;END_IF
	IF InibiscoModbusEssicatore=TRUE THEN InibiscoModbusEssicatore:=FALSE;END_IF
	NodoDaInterrogareEssicatore:=Address+1;

END_IF
END_ACTION

(* POU obj_MODBUS_Free, ST *)
FUNCTION_BLOCK obj_MODBUS_Free
(* === MODBUS PROTOCOL INTERFACE ===
   v1.1[19/06/15] - Added new VARS allocation and searching
*)
VAR CONSTANT
	VARS_Max	: BYTE := 32;
END_VAR
VAR_INPUT
	(* Settings *)
	ID			: BYTE;
	COM			: BYTE;
	BAUDRATE	: COM_BAUDRATE;
	ASCIIMODE: BOOL;

	RS485		: BOOL := FALSE;


	N_STOPBits	:BYTE:=1;

 	(* Interface *)
	MB_MASTER	: MODBUS_EXTENDED_MASTER;
	MB_Start	: BOOL;
	MB_Query	: typModbusExtendedQuery;
	MB_Resp		: typModbusResponse;
	MB_Lock		: BOOL;
	MB_timeOut	: TIME := t#500ms;

	(* Variables management *)
	VARS_En		: BOOL;
	VARS		: ARRAY [0..VARS_Max] OF typ_MODBUS_VAR;
	VARS_Check	: BOOL;
	VARS_Alarm	: BOOL;

	(* Variables allocation *)
	VAR_Pointer : POINTER TO ARRAY[0..99] OF WORD;
	VAR_Cfg		: POINTER TO typ_MODBUS_VAR;
END_VAR
VAR_OUTPUT
	(* Status *)
	Status_Log	: BYTE;
	Status_Vis	: DWORD;
END_VAR
VAR
	sta         : BYTE :=0;
	i			: BYTE;
	j			: BYTE;
	Alarm		: FLT_EVENT;
	
	VarTmr		: TON := (PT:=T#1s);
	VarSta		: BYTE; (* Status *)
	VarCnt		: BYTE; (* Scan counter *)
	VarRetry	: BYTE;
	VarAlarm	: BYTE; (* Last variable with errors *)
END_VAR
IF N_STOPBits=1 THEN MB_MASTER.csCOM_STOPBITS:=STOPBITS_1;END_IF
IF N_STOPBits=2 THEN MB_MASTER.csCOM_STOPBITS:=STOPBITS_2;END_IF

MB_MASTER(ENABLE:=TRUE,	ASCII_Mode:=ASCIIMODE, bCOM_PORT:=COM, cbCOM_BAUDRATE:=BAUDRATE,
		cfCOM_FLOW_CONTROL:=SEL(RS485,NO_FLOW_CONTROL,HALFDUPLEX),
		tTIME_OUT:=MB_timeOut,	StartFunction:=MB_Start, ExtQuery:=MB_Query, Response:=MB_Resp);

(* Process variable management *)
IF VARS_En THEN VARS_Process(); END_IF

(* Check status *)
Alarm(IN:=(MB_MASTER.bInterfaceError<>0));
IF Alarm.EVH THEN
	LogEv(SEL(MB_MASTER.bInterfaceError<>3,EL_Wrn,EL_Alarm),EO_MODBUS,ID,1,BYTE_TO_STRING(MB_MASTER.bInterfaceError));
END_IF
IF Alarm.EVL THEN								(* Trigger a fall edge: MODBUS back working *)
	LogEv(EL_Log,EO_MODBUS,ID,2,'MODBUS_OK');
END_IF

(* Log/visu status *)
   IF Alarm.IN   THEN Status_Log:=2; Status_Vis:=COLOR_RED;
ELSIF Vars_Alarm THEN Status_Log:=1; Status_Vis:=COLOR_YELLOW;
  				 ELSE Status_Log:=0; Status_Vis:=COLOR_GREEN;
END_IF
END_FUNCTION_BLOCK
ACTION VAR_Search:
(* Search VAR with specific pointer if not found return first free VAR
	[Last VAR is not active... used as safe area...] 
*)
j:=VARS_Max;
FOR i := 0 TO VARS_Max-1 DO
	IF VARS[i].Variable=0 AND j>i THEN j:=i; END_IF
	IF VARS[i].Variable=VAR_Pointer THEN
		VAR_Cfg:=ADR(VARS[i]);
		RETURN;
	END_IF
END_FOR
VAR_Cfg:=ADR(VARS[j]);
END_ACTION
ACTION VARS_Process:
(* Update var timers *)
VarTmr(IN:=(NOT VarTmr.Q));
IF VarTmr.Q THEN
	FOR i := 0 TO VARS_Max DO
		IF VARS[i].Refresh_Cnt>0 THEN VARS[i].Refresh_Cnt:=VARS[i].Refresh_Cnt-1; END_IF
	END_FOR
	VARS_Check:=TRUE;
END_IF


(* Process status *)
CASE VarSta OF
	0: (* === Init *)
		VarCnt:=0;
		VarSta:=1;

	1: (* === Wait check signal *)
		IF VARS_Check THEN				(* Decremented "Refresh_Cnt" *)
			VARS_Check:=FALSE;
			VarCnt:=0;
			VarSta:=2;
		END_IF

	2: (* === Check loop *)
		IF NOT (MB_Lock OR MB_Start) THEN
			WHILE VarCnt<=(VARS_Max-1) AND VarSta=2 DO
				(* Check only active vars *)
				IF VARS[VarCnt].Variable<>0 THEN			(* "Variable" is a pointer to word, so if 0 no address *)
					(* Check var auto-refresh on timer checks *)
					IF VARS[VarCnt].Refresh_Time>0 AND VARS[VarCnt].Refresh_Cnt=0 THEN
						VARS[VarCnt].Refresh_Cnt:=VARS[VarCnt].Refresh_Time;
						VarSta:=3;
					END_IF
					(* Check refresh for change or request *)
					CASE VARS[VarCnt].FunCode OF
						5,6,15,16: (* Write functions *)
							IF VARS[VarCnt].Variable_Size=1 THEN
								IF VARS[VarCnt].Variable^<>VARS[VarCnt].Variable_Mirror THEN
									VARS[VarCnt].Variable_Mirror:=VARS[VarCnt].Variable^;
									VarSta:=3;
								END_IF
							ELSE
								IF VARS[VarCnt].Variable_Mirror<>0 THEN
									VARS[VarCnt].Variable_Mirror:=0;
									VarSta:=3;
								END_IF
							END_IF
						1,2,3,4: (* Read functions *)
							IF VARS[VarCnt].Variable_Mirror<>0 THEN
								VARS[VarCnt].Variable_Mirror:=0;
								VarSta:=3;
							END_IF
					END_CASE
				END_IF
				(* Process query *)
				IF VarSta=3 THEN
					MB_Lock:=TRUE;
					MB_Query.SlaveAddress:=VARS[VarCnt].SlaveAddress;
					MB_Query.FunctionCode:=VARS[VarCnt].FunCode;
					CASE VARS[VarCnt].FunCode OF
						16#5,16#6,16#F,16#10:
							MB_Query.Read_Quantity:=0;
							MB_Query.Read_StartAddress:=0;
							MB_Query.Write_StartAddress:=VARS[VarCnt].FunAddress;
							MB_Query.Write_Quantity:=VARS[VarCnt].Variable_Size;
							IF VARS[VarCnt].Variable_Size=200 THEN
								COPY_32SWAP16(VARS[VarCnt].Variable, ADR(MB_Query.Write_Data[0]));
							ELSIF VARS[VarCnt].Variable_Size>1 THEN
								MEMCPY(VARS[VarCnt].Variable, ADR(MB_Query.Write_Data[0]), 2*VARS[VarCnt].Variable_Size);
							ELSE
								MB_Query.Write_Data[0]:=VARS[VarCnt].Variable^;
							END_IF
						16#1,16#2,16#3,16#4:
							MB_Query.Read_StartAddress:=VARS[VarCnt].FunAddress;
							IF VARS[VarCnt].Variable_Size=200 THEN MB_Query.Read_Quantity:=2; ELSE
							  MB_Query.Read_Quantity:=VARS[VarCnt].Variable_Size;
							END_IF
							MB_Query.Write_StartAddress:=0;
							MB_Query.Write_Quantity:=0;
					END_CASE
					VarRetry:=0;
					MB_Start:=TRUE;
				ELSE
					VarCnt:=VarCnt+1;
				END_IF
			END_WHILE
			(* Check loop completed -> no actions *)
			IF VarSta=2 THEN VarSta:=1; END_IF
		END_IF

	3: (* === Wait & process MB response *)
		IF NOT MB_Start THEN
			IF MB_MASTER.MB_Error=0 THEN
				CASE VARS[VarCnt].FunCode OF
					1,2,3,4:
						IF VARS[VarCnt].Variable_Size=200 THEN
							COPY_32SWAP16(ADR(MB_Resp.Data), VARS[VarCnt].Variable);
						ELSIF VARS[VarCnt].Variable_Size>1 THEN
							MEMCPY(ADR(MB_Resp.Data), VARS[VarCnt].Variable, 2*VARS[VarCnt].Variable_Size);
						ELSE
							VARS[VarCnt].Variable^:=MB_Resp.Data[0];
						END_IF
				END_CASE
				MB_Lock:=FALSE;
				(* Signal error recovery *)
				IF VARS_Alarm=TRUE AND VarCnt=VarAlarm THEN
					LogEv(EL_Wrn,EO_MODBUS,ID,5,'');
					VARS_Alarm:=FALSE;
				END_IF
				(* Next var *)
				VarCnt:=VarCnt+1;
				VarSta:=2;
			ELSE
				IF VarRetry<3 THEN
					VarRetry:=VarRetry+1;
					MB_Start:=TRUE;
				ELSE
					MB_Lock:=FALSE;
					(* Signal error *)
					IF VARS_Alarm=FALSE THEN
						LogEv(EL_Wrn,EO_MODBUS,ID,3,INT_TO_STRING(MB_MASTER.MB_Error));
						VARS_Alarm:=TRUE;
						VarAlarm:=VarCnt-1;
					END_IF
					(* Next var *)
					VarCnt:=VarCnt+1;
					VarSta:=2;
				END_IF
			END_IF
		END_IF

ELSE
	VarSta:=0;
END_CASE
END_ACTION

(* POU Plant_Objects/obj_MisPortata_ETH, ST *)
FUNCTION_BLOCK obj_MisPortata_ETH
(* === MODBUS-TCP PROTOCOL INTERFACE ===
   v1.0[10/06/15] - Create
*)
VAR CONSTANT
	VARS_Max	: BYTE := 32;
END_VAR
VAR_INPUT
	(* Settings *)
	ID			: BYTE;
	IP			: STRING;
	PORT		: WORD:=502;
	(* Interface *)
	MB_MASTER	: ETHERNET_MODBUSMASTER_TCP;
	MB_READBUF	: ARRAY [0..128] OF WORD;
	MB_WRITEBUF : ARRAY [0..128] OF WORD;
	MB_Start	: BOOL;
	MB_Lock		: BOOL;
	(* Variables management *)
	VARS_En		: BOOL;
	VARS		: ARRAY [0..VARS_Max] OF typ_MODBUS_VAR;
	VARS_Check	: BOOL;
	VARS_Alarm	: BOOL;
	(* Variables allocation *)
	VAR_Pointer : POINTER TO ARRAY[0..99] OF WORD;
	VAR_Cfg		: POINTER TO typ_MODBUS_VAR;
END_VAR
VAR_OUTPUT
	(* Status *)
	Status_Log	: BYTE;
	Status_Vis	: DWORD;
END_VAR
VAR
	sta         : BYTE :=0;
	i			: BYTE;
	j			: BYTE;
	Alarm		: FLT_EVENT;

	VarTmr		: TON := (PT:=T#1s);
	VarSta		: BYTE; (* Status *)
	VarCnt		: BYTE; (* Scan counter *)
	VarRetry	: BYTE;
	VarAlarm	: BYTE; (* Last variable with errors *)


	state : INT;
	ReadTmr		:	TON := (PT:=T#5s);
	retry		:	BYTE;
	retryErr	:	BYTE;
	retryErrMax	:	BYTE := 2;

	ErroreComuModBus: BOOL;
	fModbusAlr:BOOL;

	MB_RegistriHoldingLetti: ARRAY [0..300] OF WORD;

	x: INT;

	(* da diego per gestione stato stringa > 255*)
	temp :STRING(255);
	tempRaw		: ARRAY [0..MAX_SEND_TCP_CLIENT] OF BYTE;
	tempRawLen :DINT;
	longString:STRING(300);

	Parametro16:UDINT;
	Parametro17:UDINT;
	Parametro18:UDINT;
	Parametro19:UDINT;
	Parametro20:UDINT;
	Parametro21:UDINT;
	Parametro32:UDINT;
	Parametro33:UDINT;
	Parametro64:UDINT;
	Parametro65:UDINT;
	Parametro128:UDINT;

	PressioneCalcolata: REAL;
	IntPressioneCalcolata: DWORD;



	TimeOutModBus: TON;
	ErroreTimeOut: BOOL;
	test_moreno: BOOL;
	test_moreno1: WORD;
	test_moreno2: BYTE;
	AppoggioDWORD: DWORD;


	WordLW: WORD;
	WordHI: WORD;
	ValoreDWord: DWORD;
	ValoreDint: DINT;
	testINT1: DINT;
	testINT2: DINT;
END_VAR
CASE state OF
	0:	(* Refresh time manager *)
		ReadTmr(IN:=NOT ReadTmr.Q,pt:=t#1000ms);
			MB_Start:=FALSE;

		(*A tempo interrogo il nodo sempre che non ci sia qualcuno che lo sta interrogando in quel momento *)
		IF  ReadTmr.Q THEN
			state := 5;
		END_IF
	5:
	test_moreno:=MB_MASTER.xIS_CONNECTED;
	test_moreno1:=MB_MASTER.wERROR;
	test_moreno2:=MB_MASTER.bRESPONSE_UNIT_ID;
		IF  MB_MASTER.xIS_CONNECTED THEN
			state :=10;
		END_IF
	(**** Leggo le Analogiche a Disposzione  ****)

	10:	(* richiedo lettura Holding Registere   *)

			MB_MASTER.bUNIT_ID := ID;
			MB_MASTER.bFUNCTION_CODE:=3;
			MB_MASTER.wREAD_ADDRESS:=130;
			MB_MASTER.wREAD_QUANTITY:=16;
			MB_Start:=TRUE;
			state := 20;


	20:	(* Risposta all'interrogazione *)
		IF NOT MB_Start THEN
			IF MB_MASTER.wERROR<>MB_NO_ERROR THEN
				state:=300;
			ELSE

				FOR x:=0 TO MB_MASTER.wREAD_QUANTITY DO
					MB_RegistriHoldingLetti[x+MB_MASTER.wREAD_ADDRESS] := MB_READBUF[x];
				END_FOR



				WordLW:=MB_READBUF[0];
				WordHI:=MB_READBUF[1];
				(* Stabilisco il segno della variabile letta *)

				IF WordHI> 16#8000 THEN
					ValoreDWord:=16#FFFFFFFF-(WordHI*65535+WordLW);
					ValoreDint:=(DWORD_TO_DINT(ValoreDWord))*(-1);
				ELSE
					ValoreDWord:=(WordHI*65535+WordLW);
					ValoreDint:=DWORD_TO_DINT(ValoreDWord);
				END_IF;
				Parametro16:=(ValoreDint);

				WordLW:=MB_READBUF[4];
				WordHI:=MB_READBUF[5];
				(* Stabilisco il segno della variabile letta *)

				IF WordHI> 16#8000 THEN
					ValoreDWord:=16#FFFFFFFF-(WordHI*65535+WordLW);
					ValoreDint:=(DWORD_TO_DINT(ValoreDWord))*(-1);
				ELSE
					ValoreDWord:=((WordHI*65535)+WordLW);
					ValoreDint:=DWORD_TO_DINT(ValoreDWord);
				END_IF;

				Parametro18:=(ValoreDint);



(*

				AppoggioDWORD:=(MB_READBUF[1]*65535+MB_READBUF[0]);
				Parametro16:=DWORD_TO_DINT(AppoggioDWORD);
				Parametro16:=Parametro16;   (* verificato che è espresso con 2 decimali mentre al servere va 1 decimale *)
				AppoggioDWORD:=(MB_READBUF[5]*65535+MB_READBUF[4]);
				Parametro18:=DWORD_TO_DINT(AppoggioDWORD);
				Parametro18:=Parametro18;    (* verificato che è espresso con 2 decimali mentre al servere va 1 decimale *)
*)
				MB_MASTER.wREAD_ADDRESS:=180;
				MB_MASTER.wREAD_QUANTITY:=4;
				MB_Start:=TRUE;
				state := 30;

			END_IF
		END_IF

	30:	(* Risposta all'interrogazione *)
		IF NOT MB_Start THEN
			IF MB_MASTER.wERROR<>MB_NO_ERROR THEN
				state:=300;
			ELSE


				FOR x:=0 TO MB_MASTER.wREAD_QUANTITY DO
					MB_RegistriHoldingLetti[x+MB_MASTER.wREAD_ADDRESS] := MB_READBUF[x];
				END_FOR
				AppoggioDWORD:=(MB_READBUF[1]*65535+MB_READBUF[0]);
				Parametro32:=DWORD_TO_DINT(AppoggioDWORD);
				AppoggioDWORD:=(MB_READBUF[3]*65535+MB_READBUF[2]);
				Parametro33:=DWORD_TO_DINT(AppoggioDWORD);

				MB_MASTER.wREAD_ADDRESS:=230;
				MB_MASTER.wREAD_QUANTITY:=4;
				MB_Start:=TRUE;
				state := 40;

			END_IF
		END_IF

	40:	(* Risposta all'interrogazione *)
		IF NOT MB_Start THEN
			IF MB_MASTER.wERROR<>MB_NO_ERROR THEN
				state:=300;
			ELSE

				Parametro64:=MB_READBUF[1]*65535+MB_READBUF[0];
				FOR x:=0 TO MB_MASTER.wREAD_QUANTITY DO
					MB_RegistriHoldingLetti[x+MB_MASTER.wREAD_ADDRESS] := MB_READBUF[x];
				END_FOR
				MB_MASTER.wREAD_ADDRESS:=275;
				MB_MASTER.wREAD_QUANTITY:=12;
				MB_Start:=TRUE;
				state := 50;

			END_IF
		END_IF


	50:	(* Risposta all'interrogazione *)
		IF NOT MB_Start THEN
			IF MB_MASTER.wERROR<>MB_NO_ERROR THEN
				state:=300;
			ELSE

				FOR x:=0 TO MB_MASTER.wREAD_QUANTITY DO
					MB_RegistriHoldingLetti[x+MB_MASTER.wREAD_ADDRESS] := MB_READBUF[x];
				END_FOR



				WordLW:=MB_READBUF[0];
				WordHI:=MB_READBUF[1];
				(* Stabilisco il segno della variabile letta *)

				IF WordHI> 16#8000 THEN
					ValoreDWord:=16#FFFFFFFF-(WordHI*65535+WordLW);
					testINT1:=16#FFFFFFFF-((WordHI*65535)+WordLW);

					ValoreDint:=((testINT1))*(-1);
				ELSE
					ValoreDWord:=(WordHI*65535+WordLW);
					ValoreDint:=(ValoreDWord);
				END_IF;

				Parametro128:=(ValoreDint);

				MB_MASTER.wREAD_ADDRESS:=300;
				MB_MASTER.wREAD_QUANTITY:=2;
				MB_Start:=TRUE;
				state := 60;

			END_IF
		END_IF


	60:	(* Risposta all'interrogazione *)
		IF NOT MB_Start THEN
			IF MB_MASTER.wERROR<>MB_NO_ERROR THEN
				state:=300;
			ELSE

				FOR x:=0 TO MB_MASTER.wREAD_QUANTITY DO
					MB_RegistriHoldingLetti[x+MB_MASTER.wREAD_ADDRESS] := MB_READBUF[x];
				END_FOR


				state := 295;

			END_IF
		END_IF


		295:
		IF NOT MB_Start THEN
			IF  MB_MASTER.wERROR<>MB_NO_ERROR THEN (*OR ModBus.MB_MASTER.MB_Error<>0 THEN*)
				state := 300;
			ELSE
				retryErr := 0;
				retry := 0;
				state := 0;
					IF ErroreComuModBus=TRUE THEN
						LogEv(EL_Log,EO_MODBUS_TCP,ID,2,'Comunicazione_ristabilita');
						ErroreComuModBus := FALSE;
						fModbusAlr := FALSE;

				(*	WarningCtr := SEL(WarningCtr=0, WarningCtr-1, 0); *)
					END_IF
			END_IF
		END_IF



	(**** CHECK MODBUS ERROR ****)
	300: 	(* Release MODBUS *)
			retry:=retry+1;
			IF retry>3 THEN
				retry:=0;

				(* Verify if slave is dead *)
				IF retryErr < retryErrMaX THEN
					retryErr := retryErr + 1;
				ELSE
					fModbusAlr := TRUE;
					(* Verify ModBus error	*)

					IF fModbusAlr AND ErroreComuModBus=FALSE THEN
						LogEv(SEL(MB_MASTER.wERROR>0,EL_Wrn,EL_Alarm),EO_MODBUS_TCP,ID,1,WORD_TO_STRING(MB_MASTER.wERROR));
						ErroreComuModBus := TRUE;
					END_IF
				END_IF

				END_IF
			state:=0;
END_CASE



MB_MASTER( strIP_ADDRESS:=IP, wPORT:=PORT, tTIME_OUT:=T#750MS, (*xCONNECT:=TRUE,*)
		   ptREAD_DATA:=ADR(MB_READBUF), ptSEND_DATA:=ADR(MB_WRITEBUF), xSEND:=MB_Start );

IF state<>0 THEN
	MB_MASTER.xCONNECT:=TRUE;
ELSE
	MB_MASTER.xCONNECT:=FALSE;
END_IF
(*
(* Process variable management *)
IF VARS_En THEN VARS_Process(); END_IF
*)

(* Controllo Time Out Ciclo ModBus *)

TimeOutModBus(In:=state<>0,PT:=t#5s);
IF TimeOutModBus.Q THEN
	State:=300;
END_IF


(* Log/visu status *)
   IF Alarm.IN   THEN Status_Log:=2; Status_Vis:=COLOR_RED;
ELSIF Vars_Alarm OR ErroreComuModBus  THEN
	Status_Log:=1; Status_Vis:=COLOR_YELLOW;
  ELSE
	Status_Log:=0; Status_Vis:=COLOR_GREEN;
END_IF
END_FUNCTION_BLOCK
ACTION AddLogData:
Logger.s1:=CONCAT('&','FPT');
IF ID<10 THEN Logger.s1:=CONCAT(Logger.s1,'0');END_IF
Logger.s1:=CONCAT(Logger.s1,BYTE_TO_STRING(ID));
Logger.s1:=CONCAT(Logger.s1,'=');


FOR tempRawLen:=0 TO MAX_SEND_TCP_CLIENT DO
                tempRaw[tempRawLen]:=0;
END_FOR

tempRawLen:=0;


temp:=Logger.s1;
ADDSTRING(ADR(tempRaw), ADR(temp), tempRawLen);

temp:=CONCAT(WORD_TO_STRING(Status_Log),';'); (*1*)
ADDSTRING(ADR(tempRaw), ADR(temp), tempRawLen);

temp:=CONCAT(DWORD_TO_STRING(Parametro16),';'); (*2*)
ADDSTRING(ADR(tempRaw), ADR(temp), tempRawLen);


temp:=CONCAT(DINT_TO_STRING(Parametro18),';'); (*3*)
ADDSTRING(ADR(tempRaw), ADR(temp), tempRawLen);


(* calcolo per passsare la pressione partendo dal psi *)
PressioneCalcolata:=DWORD_TO_REAL(parametro33)*0.068949; (*4*)
IntPressioneCalcolata:=parametro32;
temp:=CONCAT(DWORD_TO_STRING(Parametro32),';');
ADDSTRING(ADR(tempRaw), ADR(temp), tempRawLen)
;
temp:=CONCAT(DWORD_TO_STRING(Parametro64),';'); (*5*)
ADDSTRING(ADR(tempRaw), ADR(temp), tempRawLen);

temp:=DWORD_TO_STRING(Parametro128); (*6*)
ADDSTRING(ADR(tempRaw), ADR(temp), tempRawLen);



ADDSTRING(ADR(Logger.TData), ADR(tempRaw), Logger.TLen);
END_ACTION
ACTION VAR_Search:
(* Search VAR with specific pointer if not found return first free VAR
	[Last VAR is not active... used as safe area...] 
*)
j:=VARS_Max;
FOR i := 0 TO VARS_Max-1 DO
	IF VARS[i].Variable=0 AND j>i THEN j:=i; END_IF
	IF VARS[i].Variable=VAR_Pointer THEN
		VAR_Cfg:=ADR(VARS[i]);
		RETURN;
	END_IF
END_FOR
VAR_Cfg:=ADR(VARS[j]);
END_ACTION
ACTION VARS_Process:
(* Update var timers *)
VarTmr(IN:=(NOT VarTmr.Q));
IF VarTmr.Q THEN
	FOR i := 0 TO VARS_Max DO
		IF VARS[i].Refresh_Cnt>0 THEN VARS[i].Refresh_Cnt:=VARS[i].Refresh_Cnt-1; END_IF
	END_FOR
	VARS_Check:=TRUE;
END_IF


(* Process status *)
CASE VarSta OF
	0: (* === Init *)
		VarCnt:=0;
		VarSta:=1;

	1: (* === Wait check signal *)
		IF VARS_Check THEN
			VARS_Check:=FALSE;
			VarCnt:=0;
			VarSta:=2;
		END_IF

	2: (* === Check loop *)
		IF NOT (MB_Lock OR MB_Start) THEN
			WHILE VarCnt<=(VARS_Max-1) AND VarSta=2 DO
				(* Check only active vars *)
				IF VARS[VarCnt].Variable<>0 THEN
					(* Check var auto-refresh on timer checks *)
					IF VARS[VarCnt].Refresh_Time>0 AND VARS[VarCnt].Refresh_Cnt=0 THEN
						VARS[VarCnt].Refresh_Cnt:=VARS[VarCnt].Refresh_Time;
						VarSta:=3;
					END_IF
					(* Check refresh for change or request *)
					CASE VARS[VarCnt].FunCode OF
						5,6,15,16: (* Write functions *)
							IF VARS[VarCnt].Variable_Size=1 THEN
								IF VARS[VarCnt].Variable^<>VARS[VarCnt].Variable_Mirror THEN
									VARS[VarCnt].Variable_Mirror:=VARS[VarCnt].Variable^;
									VarSta:=3;
								END_IF
							ELSE
								IF VARS[VarCnt].Variable_Mirror<>0 THEN
									VARS[VarCnt].Variable_Mirror:=0;
									VarSta:=3;
								END_IF
							END_IF
						1,2,3,4: (* Write functions *)
							IF VARS[VarCnt].Variable_Mirror<>0 THEN
								VARS[VarCnt].Variable_Mirror:=0;
								VarSta:=3;
							END_IF
					END_CASE
				END_IF
				(* Process query *)
				IF VarSta=3 THEN
					MB_Lock:=TRUE;
					MB_MASTER.bUNIT_ID:=VARS[VarCnt].SlaveAddress;
					MB_MASTER.bFUNCTION_CODE:=VARS[VarCnt].FunCode;
					CASE VARS[VarCnt].FunCode OF
						16#5,16#6,16#F,16#10:
							MB_MASTER.wREAD_ADDRESS:=0;
							MB_MASTER.wREAD_QUANTITY:=0;
							MB_MASTER.wWRITE_ADDRESS:=VARS[VarCnt].FunAddress;
							MB_MASTER.wWRITE_QUANTITY:=VARS[VarCnt].Variable_Size;
							IF VARS[VarCnt].Variable_Size=200 THEN
								COPY_32SWAP16(VARS[VarCnt].Variable, ADR(MB_WRITEBUF));
							ELSIF VARS[VarCnt].Variable_Size>1 THEN
								MEMCPY(VARS[VarCnt].Variable, ADR(MB_WRITEBUF), 2*VARS[VarCnt].Variable_Size);
							ELSE
								MB_WRITEBUF[0]:=VARS[VarCnt].Variable^;
							END_IF
						16#1,16#2,16#3,16#4:
							MB_MASTER.wREAD_ADDRESS:=VARS[VarCnt].FunAddress;
							IF VARS[VarCnt].Variable_Size=200 THEN MB_MASTER.wREAD_QUANTITY:=2; ELSE
							  MB_MASTER.wREAD_QUANTITY:=VARS[VarCnt].Variable_Size;
							END_IF
							MB_MASTER.wWRITE_ADDRESS:=0;
							MB_MASTER.wWRITE_QUANTITY:=0;
					END_CASE
					VarRetry:=0;
					MB_Start:=TRUE;
				ELSE
					VarCnt:=VarCnt+1;
				END_IF
			END_WHILE
			(* Check loop completed -> no actions *)
			IF VarSta=2 THEN VarSta:=1; END_IF
		END_IF

	3: (* === Wait & process MB response *)
		IF NOT MB_Start THEN
			IF MB_MASTER.wERROR=0 THEN
				CASE VARS[VarCnt].FunCode OF
					1,2,3,4:
						IF VARS[VarCnt].Variable_Size=200 THEN
							COPY_32SWAP16(ADR(MB_READBUF), VARS[VarCnt].Variable);
						ELSIF VARS[VarCnt].Variable_Size>1 THEN
							MEMCPY(ADR(MB_READBUF), VARS[VarCnt].Variable, 2*VARS[VarCnt].Variable_Size);
						ELSE
							VARS[VarCnt].Variable^:=MB_READBUF[0];
						END_IF
				END_CASE
				MB_Lock:=FALSE;
				(* Signal error recovery *)
				IF VARS_Alarm=TRUE AND VarCnt=VarAlarm THEN
					LogEv(EL_Wrn,EO_MODBUS_TCP,ID,5,'');
					VARS_Alarm:=FALSE;
				END_IF
				(* Next var *)
				VarCnt:=VarCnt+1;
				VarSta:=2;
			ELSE
				IF VarRetry<10 THEN
					VarRetry:=VarRetry+1;
					MB_Start:=TRUE;
				ELSE
					MB_Lock:=FALSE;
					(* Signal error *)
					IF VARS_Alarm=FALSE THEN
						LogEv(EL_Wrn,EO_MODBUS_TCP,ID,3,WORD_TO_STRING(MB_MASTER.wERROR));
						VARS_Alarm:=TRUE;
						VarAlarm:=VarCnt-1;
					END_IF
					(* Next var *)
					VarCnt:=VarCnt+1;
					VarSta:=2;
				END_IF
			END_IF
		END_IF

ELSE
	VarSta:=0;
END_CASE
END_ACTION

(* POU Plant_Objects/obj_MisPortata_MB, ST *)
FUNCTION_BLOCK obj_MisPortata_MB
VAR CONSTANT
	TimeOutModBus: TON;
END_VAR
VAR_INPUT
	ID			:	BYTE;
	Address		:	BYTE;

	(* Modbus *)
	Refresh_Now	:	BOOL;			(* Richiesta di lettura stato macchina Immediata  *)
	retryErrMax	:	BYTE := 2;

	OnOff		: 	BOOL;

	IndirizzoDaScrivere: WORD;
	DatoDaScrivere: INT;
	ScriviDato: BOOL;
	ScriviCoil: BOOL;

	fWriteAttivazioneComandi:BOOL;

END_VAR
VAR_IN_OUT
	ModBus		:obj_MODBUS;
END_VAR
VAR_OUTPUT
	Run			:	BOOL;

	Status_Log	:	WORD;
	Status_Vis	:	DWORD;
END_VAR
VAR
	(* da diego per gestione stato stringa > 255*)
	temp :STRING(255);
	tempRaw		: ARRAY [0..MAX_SEND_TCP_CLIENT] OF BYTE;
	tempRawLen :DINT;
	longString:STRING(255);

	(* Timer manage switch on/off delay *)
	Delay		: 	TONOF;
	Warning		:	FLT_TAP := (TAP:=100);

	state		:	INT;
	retry		:	BYTE;
	retryErr	:	BYTE;
	ReadTmr		:	TON := (PT:=T#5s);
	fModbusAlr:BOOL;



	VerificaFuctionCode: INT;
	VerificaNodoLetto: INT;
	ErroreComuModBus: BOOL;
	IndiceErrore: BYTE;

(*	MB_BitStato: ARRAY [0..1] OF BOOL;
	MB_RegistriLetti: ARRAY [0..1] OF INT;
	MB_RegistriHoldingLetti: ARRAY [0..255] OF WORD;
	MB_BitStatoCoil: ARRAY [0..1] OF BOOL; *)


	Parametro16:DWORD;
	Parametro17:DWORD;
	Parametro18:DWORD;
	Parametro19:DWORD;
	Parametro20:DWORD;
	Parametro21:DWORD;
	Parametro32:DWORD;
	Parametro33:DWORD;
	Parametro64:DWORD;
	Parametro65:DWORD;
	Parametro128:DWORD;





	AddressRead: BYTE;
	index: BYTE;
	indexErr: BYTE;





	x: INT;

	PressioneCalcolata: REAL;
	IntPressioneCalcolata: INT;
	Parametro128_1: WORD;
	Parametro128_2: WORD;
	Parametro128_3: WORD;
	Parametro128_4: WORD;
	WordLW: WORD;
	WordHI: WORD;
	ValoreDint: DINT;
	ValoreDWord: DWORD;
END_VAR
(* Call ModBus state machine *)
Stm();


(* Seganalzione stato Compressore  *)
IF ErroreComuModBus THEN
		Status_Log:=2; Status_Vis:=16#2020F0;
(*	ELSIF Warning OR Warning2 THEN
		Status_Log:=1; Status_Vis:=16#20F0F0; *)
    ELSE
		Status_Log:=0;
		Status_Vis:=16#006000;
END_IF
END_FUNCTION_BLOCK
ACTION AddLogData:
Logger.s1:=INSERT('&FPT=',BYTE_TO_STRING(ID),4);
IF ID<10 THEN Logger.s1:=INSERT(Logger.s1,'0',4); END_IF

FOR tempRawLen:=0 TO MAX_SEND_TCP_CLIENT DO
                tempRaw[tempRawLen]:=0;
END_FOR

tempRawLen:=0;


temp:=Logger.s1;
ADDSTRING(ADR(tempRaw), ADR(temp), tempRawLen);

temp:=CONCAT(WORD_TO_STRING(Status_Log),';');
ADDSTRING(ADR(tempRaw), ADR(temp), tempRawLen); (*1 param*)

temp:=CONCAT(DWORD_TO_STRING(Parametro16),';');
ADDSTRING(ADR(tempRaw), ADR(temp), tempRawLen);(* 2 param *)


temp:=CONCAT(DWORD_TO_STRING(Parametro17*10),';');   (* ora l-min poi si dovra mettere par17 *)
ADDSTRING(ADR(tempRaw), ADR(temp), tempRawLen);(* 3 param *)


(* calcolo per passsare la pressione partendo dal psi *)
PressioneCalcolata:=DWORD_TO_REAL(parametro33)*0.068949;
IntPressioneCalcolata:=REAL_TO_INT(PressioneCalcolata*10);

temp:=CONCAT(DINT_TO_STRING(IntPressioneCalcolata),';'); (* 4 param *)
ADDSTRING(ADR(tempRaw), ADR(temp), tempRawLen);

temp:=CONCAT(DWORD_TO_STRING(Parametro64),';');
ADDSTRING(ADR(tempRaw), ADR(temp), tempRawLen); (* 5 param*)

temp:=DWORD_TO_STRING(Parametro128);
ADDSTRING(ADR(tempRaw), ADR(temp), tempRawLen); (* 6 param*)



ADDSTRING(ADR(Logger.TData), ADR(tempRaw), Logger.TLen);
END_ACTION
ACTION Stm:
CASE state OF
	0:	(* Refresh time manager *)
		ReadTmr(IN:=NOT ReadTmr.Q);
		(*A tempo interrogo il nodo sempre che non ci sia qualcuno che lo sta interrogando in quel momento *)

		IF (ReadTmr.Q AND NodoDaInterrogareMisuratoreDiPortata=Address ) OR Refresh_Now AND NOT InibiscoModbusMisuratoreDiPortata THEN
			state := 10;
			ReadTmr.PT := T#500ms;  (* moreno *)
			Refresh_Now := FALSE;
			InibiscoModbusMisuratoreDiPortata := TRUE;
		END_IF

	(**** Leggo le Analogiche a Disposzione  ****)

	10:	(* richiedo lettura Holding Registere   *)

		Modbus.MB_Query.SlaveAddress := Address;
		Modbus.MB_Query.FunctionCode := 3;
		ModBus.MB_Query.Read_StartAddress := 16; (* 41 ; *)
		ModBus.MB_Query.Read_Quantity :=2;
		ModBus.MB_Start := TRUE;
		state := 20;

	20:	(* Risposta all'interrogazione *)
		IF NOT ModBus.MB_Start   THEN
			VerificaFuctionCode:=ModBus.MB_Resp.FunctionCode;
			VerificaNodoLetto:=ModBus.MB_Resp.SlaveAddress;

			IF ModBus.MB_MASTER.MB_Error<>0 THEN
				state := 300;
			ELSE
			(*	FOR x:=0 TO ModBus.MB_Query.Read_Quantity DO
					MB_RegistriHoldingLetti[x+ModBus.MB_Query.Read_StartAddress] := ModBus.MB_Resp.Data[x];   	(* Vedi tabella *)
				END_FOR *)


				WordLW:=ModBus.MB_Resp.Data[0];
				WordHI:=ModBus.MB_Resp.Data[1];
				(* Stabilisco il segno della variabile letta *)

				IF WordHI> 16#8000 THEN
					ValoreDWord:=16#FFFFFFFF-(WordHI*65536+WordLW);
					ValoreDint:=(DWORD_TO_DINT(ValoreDWord))*(-1);
				ELSE
					ValoreDWord:=(WordHI*65536+WordLW);
					ValoreDint:=DWORD_TO_DINT(ValoreDWord);
				END_IF;







				Parametro16:=ModBus.MB_Resp.Data[1]*65535+ModBus.MB_Resp.Data[0];


				ModBus.MB_Query.Read_StartAddress :=17; 	(* richiedo lettura altri Parametri *)
				ModBus.MB_Query.Read_Quantity := 2;
				ModBus.MB_Start := TRUE;

				state := 30;
			END_IF
		END_IF

	30: (* Rispota Altri paramenti *)
		IF NOT ModBus.MB_Start  THEN

			IF ModBus.MB_MASTER.MB_Error<>0 THEN
				state := 300;
			ELSE

			(*	FOR x:=0 TO ModBus.MB_Query.Read_Quantity DO
					MB_RegistriHoldingLetti[x+ModBus.MB_Query.Read_StartAddress] := ModBus.MB_Resp.Data[x];   	(* Vedi tabella *)
				END_FOR *)


				Parametro17:=ModBus.MB_Resp.Data[1]*65535+ModBus.MB_Resp.Data[0];


				ModBus.MB_Query.Read_StartAddress :=18; 	(* richiedo lettura altri Parametri *)
				ModBus.MB_Query.Read_Quantity := 2;
				ModBus.MB_Start := TRUE;

				state := 40;
			END_IF
		END_IF


	40: (* Rispota Altri paramenti *)
		IF NOT ModBus.MB_Start  THEN

			IF ModBus.MB_MASTER.MB_Error<>0 THEN
				state := 300;
			ELSE

			(*	FOR x:=0 TO ModBus.MB_Query.Read_Quantity DO
					MB_RegistriHoldingLetti[x+ModBus.MB_Query.Read_StartAddress] := ModBus.MB_Resp.Data[x];   	(* Vedi tabella *)
				END_FOR *)



				Parametro18:=ModBus.MB_Resp.Data[1]*65535+ModBus.MB_Resp.Data[0];


				ModBus.MB_Query.Read_StartAddress :=19; 	(* richiedo lettura altri Parametri *)
				ModBus.MB_Query.Read_Quantity := 2;
				ModBus.MB_Start := TRUE;

				state := 50;
			END_IF
		END_IF

	50: (* Rispota Altri paramenti *)
		IF NOT ModBus.MB_Start  THEN

			IF ModBus.MB_MASTER.MB_Error<>0 THEN
				state := 300;
			ELSE

			(*	FOR x:=0 TO ModBus.MB_Query.Read_Quantity DO
					MB_RegistriHoldingLetti[x+ModBus.MB_Query.Read_StartAddress] := ModBus.MB_Resp.Data[x];   	(* Vedi tabella *)
				END_FOR *)


				Parametro19:=ModBus.MB_Resp.Data[1]*65535+ModBus.MB_Resp.Data[0];


				ModBus.MB_Query.Read_StartAddress :=20; 	(* richiedo lettura altri Parametri *)
				ModBus.MB_Query.Read_Quantity := 2;
				ModBus.MB_Start := TRUE;

				state := 60;
			END_IF
		END_IF

	60: (* Rispota Altri paramenti *)
		IF NOT ModBus.MB_Start  THEN

			IF ModBus.MB_MASTER.MB_Error<>0 THEN
				state := 300;
			ELSE

			(*	FOR x:=0 TO ModBus.MB_Query.Read_Quantity DO
					MB_RegistriHoldingLetti[x+ModBus.MB_Query.Read_StartAddress] := ModBus.MB_Resp.Data[x];   	(* Vedi tabella *)
				END_FOR *)


				Parametro20:=ModBus.MB_Resp.Data[1]*65535+ModBus.MB_Resp.Data[0];


				ModBus.MB_Query.Read_StartAddress :=21; 	(* richiedo lettura altri Parametri *)
				ModBus.MB_Query.Read_Quantity := 2;
				ModBus.MB_Start := TRUE;

				state := 70;
			END_IF
		END_IF

	70: (* Rispota Altri paramenti *)
		IF NOT ModBus.MB_Start  THEN

			IF ModBus.MB_MASTER.MB_Error<>0 THEN
				state := 300;
			ELSE

			(*	FOR x:=0 TO ModBus.MB_Query.Read_Quantity DO
					MB_RegistriHoldingLetti[x+ModBus.MB_Query.Read_StartAddress] := ModBus.MB_Resp.Data[x];   	(* Vedi tabella *)
				END_FOR *)


				Parametro21:=ModBus.MB_Resp.Data[1]*65535+ModBus.MB_Resp.Data[0];


				ModBus.MB_Query.Read_StartAddress :=32; 	(* richiedo lettura altri Parametri *)
				ModBus.MB_Query.Read_Quantity := 2;
				ModBus.MB_Start := TRUE;

				state := 80;
			END_IF
		END_IF

	80: (* Rispota Altri paramenti *)
		IF NOT ModBus.MB_Start  THEN

			IF ModBus.MB_MASTER.MB_Error<>0 THEN
				state := 300;
			ELSE

			(*	FOR x:=0 TO ModBus.MB_Query.Read_Quantity DO
					MB_RegistriHoldingLetti[x+ModBus.MB_Query.Read_StartAddress] := ModBus.MB_Resp.Data[x];   	(* Vedi tabella *)
				END_FOR *)


				Parametro32:=ModBus.MB_Resp.Data[1]*65535+ModBus.MB_Resp.Data[0];


				ModBus.MB_Query.Read_StartAddress :=33; 	(* richiedo lettura altri Parametri *)
				ModBus.MB_Query.Read_Quantity := 2;
				ModBus.MB_Start := TRUE;

				state := 90;
			END_IF
		END_IF

	90: (* Rispota Altri paramenti *)
		IF NOT ModBus.MB_Start  THEN

			IF ModBus.MB_MASTER.MB_Error<>0 THEN
				state := 300;
			ELSE

			(*	FOR x:=0 TO ModBus.MB_Query.Read_Quantity DO
					MB_RegistriHoldingLetti[x+ModBus.MB_Query.Read_StartAddress] := ModBus.MB_Resp.Data[x];   	(* Vedi tabella *)
				END_FOR *)


				Parametro33:=ModBus.MB_Resp.Data[1]*65535+ModBus.MB_Resp.Data[0];


				ModBus.MB_Query.Read_StartAddress :=64; 	(* richiedo lettura altri Parametri *)
				ModBus.MB_Query.Read_Quantity := 2;
				ModBus.MB_Start := TRUE;

				state :=100;
			END_IF
		END_IF

	100: (* Rispota Altri paramenti *)
		IF NOT ModBus.MB_Start  THEN

			IF ModBus.MB_MASTER.MB_Error<>0 THEN
				state := 300;
			ELSE

			(*	FOR x:=0 TO ModBus.MB_Query.Read_Quantity DO
					MB_RegistriHoldingLetti[x+ModBus.MB_Query.Read_StartAddress] := ModBus.MB_Resp.Data[x];   	(* Vedi tabella *)
				END_FOR *)


				Parametro64:=ModBus.MB_Resp.Data[1]*65535+ModBus.MB_Resp.Data[0];


				ModBus.MB_Query.Read_StartAddress :=65; 	(* richiedo lettura altri Parametri *)
				ModBus.MB_Query.Read_Quantity := 2;
				ModBus.MB_Start := TRUE;

				state := 110;
			END_IF
		END_IF

	110: (* Rispota Altri paramenti *)
		IF NOT ModBus.MB_Start  THEN

			IF ModBus.MB_MASTER.MB_Error<>0 THEN
				state := 300;
			ELSE

			(*	FOR x:=0 TO ModBus.MB_Query.Read_Quantity DO
					MB_RegistriHoldingLetti[x+ModBus.MB_Query.Read_StartAddress] := ModBus.MB_Resp.Data[x];   	(* Vedi tabella *)
				END_FOR *)


				Parametro65:=ModBus.MB_Resp.Data[1]*65535+ModBus.MB_Resp.Data[0];


				ModBus.MB_Query.Read_StartAddress :=128; 	(* richiedo lettura altri Parametri *)
				ModBus.MB_Query.Read_Quantity := 2;
				ModBus.MB_Start := TRUE;

				state := 120;
			END_IF
		END_IF

	120: (* Rispota Altri paramenti *)
		IF NOT ModBus.MB_Start  THEN

			IF ModBus.MB_MASTER.MB_Error<>0 THEN
				state := 300;
			ELSE

			(*	FOR x:=0 TO ModBus.MB_Query.Read_Quantity DO
					MB_RegistriHoldingLetti[x+ModBus.MB_Query.Read_StartAddress] := ModBus.MB_Resp.Data[x];   	(* Vedi tabella *)
				END_FOR *)

				Parametro128_1:=ModBus.MB_Resp.Data[0];
				Parametro128_2:=ModBus.MB_Resp.Data[1];
				Parametro128_3:=ModBus.MB_Resp.Data[2];
				Parametro128_4:=ModBus.MB_Resp.Data[3];

				Parametro128:=ModBus.MB_Resp.Data[1]*65535+ModBus.MB_Resp.Data[0];


				state :=295;
			END_IF
		END_IF


(*




	290:    (* Scrittura BOOL - COIL o WORD *)
		IF NOT ModBus.MB_Start THEN
			IF ModBus.MB_MASTER.MB_Error<>0 THEN (*OR ModBus.MB_MASTER.MB_Error<>0 THEN*)
				state := 300;
			ELSE
				IF ScriviDato THEN
					IF ScriviCoil THEN
						Modbus.MB_Query.FunctionCode := 5;
					ELSE
						Modbus.MB_Query.FunctionCode := 6;
					END_IF
					Modbus.MB_Query.SlaveAddress := Address;
					ModBus.MB_Query.Write_StartAddress := IndirizzoDaScrivere;
					ModBus.MB_Query.Write_Quantity :=1;
					ModBus.MB_Query.Write_Data[0] := DatoDaScrivere;
					ModBus.MB_Start := TRUE;
						IF ScriviCoil THEN
							IF 	MB_BitStato[IndirizzoDaScrivere]=WORD_TO_BOOL(DatoDaScrivere-1) THEN
								ScriviDato:=FALSE;
							END_IF
						ELSE
							IF 	MB_RegistriLetti[IndirizzoDaScrivere]=DatoDaScrivere THEN
								ScriviDato:=FALSE;
							END_IF
						END_IF
					state := 295;
				ELSE
					state := 295;
				END_IF
			END_IF
		END_IF


*)

		295:
		IF NOT ModBus.MB_Start THEN
			IF ModBus.MB_MASTER.MB_Error<>0 THEN (*OR ModBus.MB_MASTER.MB_Error<>0 THEN*)
				state := 300;
			ELSE
				IF fModbusAlr THEN fModbusAlr := FALSE; END_IF
				NodoDaInterrogareMisuratoreDiPortata:=Address+1;
				InibiscoModbusMisuratoreDiPortata:=FALSE;
				retryErr := 0;
				retry := 0;
				state := 0;
					IF fModbusAlr=FALSE AND ErroreComuModBus=TRUE THEN
						LogEv(EL_Log,EO_FPT,ID,62,'ComunicazioneModBus_OK');
						ErroreComuModBus := FALSE;
				(*	WarningCtr := SEL(WarningCtr=0, WarningCtr-1, 0); *)
					END_IF


			END_IF
		END_IF



	(**** CHECK MODBUS ERROR ****)
	300: 	(* Release MODBUS *)
			InibiscoModbusMisuratoreDiPortata:=FALSE;
			(* Retries *)
			retry:=retry+1;
			IF retry>3 THEN
				retry:=0;

				(* Verify if slave is dead *)
				IF retryErr < retryErrMaX THEN
					retryErr := retryErr + 1;
				ELSE
					fModbusAlr := TRUE;
					(* Verify ModBus error	*)

					IF fModbusAlr AND ErroreComuModBus=FALSE THEN
						LogEv(EL_Alarm,EO_FPT,ID,61,CONCAT('ErroreModbus_',INT_TO_STRING(ModBus.MB_MASTER.MB_Error)));
						ErroreComuModBus := TRUE;
					END_IF
				END_IF

				END_IF
			Refresh_Now := FALSE;
			NodoDaInterrogareMisuratoreDiPortata:=Address+1;
			state:=0;
END_CASE


(* calcolo per passsare la pressione partendo dal psi *)
PressioneCalcolata:=DWORD_TO_REAL(parametro33)*0.06895;
IntPressioneCalcolata:=REAL_TO_INT(PressioneCalcolata*10);



(* Controllo Time Out Ciclo ModBus *)

TimeOutModBus(In:=state<>0,PT:=t#30s);
IF TimeOutModBus.Q THEN
	State:=0;
	(*Refresh_Now:=TRUE;  (* Rilancio la lettura del nodo *) *)
	IF MODBUS.MB_Lock=TRUE THEN MODBUS.MB_Lock:=FALSE;END_IF
	IF InibiscoModbusMisuratoreDiPortata=TRUE THEN InibiscoModbusMisuratoreDiPortata:=FALSE;END_IF
	NodoDaInterrogareMisuratoreDiPortata:=Address+1;

END_IF
END_ACTION

(* POU Plant_Objects/obj_MODBUS_TCP, ST *)
FUNCTION_BLOCK obj_MODBUS_TCP
(* === MODBUS-TCP PROTOCOL INTERFACE ===
   v1.0[10/06/15] - Create
*)
VAR CONSTANT
	VARS_Max	: BYTE := 32;
END_VAR
VAR_INPUT
	(* Settings *)
	ID			: BYTE;
	IP			: STRING;
	PORT		: WORD:=502;
	(* Interface *)
	MB_MASTER	: ETHERNET_MODBUSMASTER_TCP;
	MB_READBUF	: ARRAY [0..128] OF WORD;
	MB_WRITEBUF : ARRAY [0..128] OF WORD;
	MB_Start	: BOOL;
	MB_Lock		: BOOL;
	(* Variables management *)
	VARS_En		: BOOL;
	VARS		: ARRAY [0..VARS_Max] OF typ_MODBUS_VAR;
	VARS_Check	: BOOL;
	VARS_Alarm	: BOOL;
	(* Variables allocation *)
	VAR_Pointer : POINTER TO ARRAY[0..99] OF WORD;
	VAR_Cfg		: POINTER TO typ_MODBUS_VAR;
END_VAR
VAR_OUTPUT
	(* Status *)
	Status_Log	: BYTE;
	Status_Vis	: DWORD;
END_VAR
VAR
	sta         : BYTE :=0;
	i			: BYTE;
	j			: BYTE;
	Alarm		: FLT_EVENT;

	VarTmr		: TON := (PT:=T#1s);
	VarSta		: BYTE; (* Status *)
	VarCnt		: BYTE; (* Scan counter *)
	VarRetry	: BYTE;
	VarAlarm	: BYTE; (* Last variable with errors *)
END_VAR
MB_MASTER( strIP_ADDRESS:=IP, wPORT:=PORT, tTIME_OUT:=T#750MS, (*xCONNECT:=TRUE,*)
		   ptREAD_DATA:=ADR(MB_READBUF), ptSEND_DATA:=ADR(MB_WRITEBUF), xSEND:=MB_Start );

IF sta=0 THEN
	MB_MASTER.xCONNECT:=TRUE;
	sta:=1;
END_IF

(* Process variable management *)
IF VARS_En THEN VARS_Process(); END_IF

(* Check status *)
Alarm(IN:=(MB_MASTER.wERROR<>0));
IF Alarm.EVH THEN
	LogEv(SEL(MB_MASTER.wERROR>0,EL_Wrn,EL_Alarm),EO_MODBUS_TCP,ID,1,WORD_TO_STRING(MB_MASTER.wERROR));
END_IF
IF Alarm.EVL THEN
	LogEv(EL_Log,EO_MODBUS_TCP,ID,2,'');
END_IF

(* Log/visu status *)
   IF Alarm.IN   THEN Status_Log:=2; Status_Vis:=COLOR_RED;
ELSIF Vars_Alarm THEN Status_Log:=1; Status_Vis:=COLOR_YELLOW;
  				 ELSE Status_Log:=0; Status_Vis:=COLOR_GREEN;
END_IF
END_FUNCTION_BLOCK
ACTION VAR_Search:
(* Search VAR with specific pointer if not found return first free VAR
	[Last VAR is not active... used as safe area...] 
*)
j:=VARS_Max;
FOR i := 0 TO VARS_Max-1 DO
	IF VARS[i].Variable=0 AND j>i THEN j:=i; END_IF
	IF VARS[i].Variable=VAR_Pointer THEN
		VAR_Cfg:=ADR(VARS[i]);
		RETURN;
	END_IF
END_FOR
VAR_Cfg:=ADR(VARS[j]);
END_ACTION
ACTION VARS_Process:
(* Update var timers *)
VarTmr(IN:=(NOT VarTmr.Q));
IF VarTmr.Q THEN
	FOR i := 0 TO VARS_Max DO
		IF VARS[i].Refresh_Cnt>0 THEN VARS[i].Refresh_Cnt:=VARS[i].Refresh_Cnt-1; END_IF
	END_FOR
	VARS_Check:=TRUE;
END_IF


(* Process status *)
CASE VarSta OF
	0: (* === Init *)
		VarCnt:=0;
		VarSta:=1;

	1: (* === Wait check signal *)
		IF VARS_Check THEN
			VARS_Check:=FALSE;
			VarCnt:=0;
			VarSta:=2;
		END_IF

	2: (* === Check loop *)
		IF NOT (MB_Lock OR MB_Start) THEN
			WHILE VarCnt<=(VARS_Max-1) AND VarSta=2 DO
				(* Check only active vars *)
				IF VARS[VarCnt].Variable<>0 THEN
					(* Check var auto-refresh on timer checks *)
					IF VARS[VarCnt].Refresh_Time>0 AND VARS[VarCnt].Refresh_Cnt=0 THEN
						VARS[VarCnt].Refresh_Cnt:=VARS[VarCnt].Refresh_Time;
						VarSta:=3;
					END_IF
					(* Check refresh for change or request *)
					CASE VARS[VarCnt].FunCode OF
						5,6,15,16: (* Write functions *)
							IF VARS[VarCnt].Variable_Size=1 THEN
								IF VARS[VarCnt].Variable^<>VARS[VarCnt].Variable_Mirror THEN
									VARS[VarCnt].Variable_Mirror:=VARS[VarCnt].Variable^;
									VarSta:=3;
								END_IF
							ELSE
								IF VARS[VarCnt].Variable_Mirror<>0 THEN
									VARS[VarCnt].Variable_Mirror:=0;
									VarSta:=3;
								END_IF
							END_IF
						1,2,3,4: (* Write functions *)
							IF VARS[VarCnt].Variable_Mirror<>0 THEN
								VARS[VarCnt].Variable_Mirror:=0;
								VarSta:=3;
							END_IF
					END_CASE
				END_IF
				(* Process query *)
				IF VarSta=3 THEN
					MB_Lock:=TRUE;
					MB_MASTER.bUNIT_ID:=VARS[VarCnt].SlaveAddress;
					MB_MASTER.bFUNCTION_CODE:=VARS[VarCnt].FunCode;
					CASE VARS[VarCnt].FunCode OF
						16#5,16#6,16#F,16#10:
							MB_MASTER.wREAD_ADDRESS:=0;
							MB_MASTER.wREAD_QUANTITY:=0;
							MB_MASTER.wWRITE_ADDRESS:=VARS[VarCnt].FunAddress;
							MB_MASTER.wWRITE_QUANTITY:=VARS[VarCnt].Variable_Size;
							IF VARS[VarCnt].Variable_Size=200 THEN
								COPY_32SWAP16(VARS[VarCnt].Variable, ADR(MB_WRITEBUF));
							ELSIF VARS[VarCnt].Variable_Size>1 THEN
								MEMCPY(VARS[VarCnt].Variable, ADR(MB_WRITEBUF), 2*VARS[VarCnt].Variable_Size);
							ELSE
								MB_WRITEBUF[0]:=VARS[VarCnt].Variable^;
							END_IF
						16#1,16#2,16#3,16#4:
							MB_MASTER.wREAD_ADDRESS:=VARS[VarCnt].FunAddress;
							IF VARS[VarCnt].Variable_Size=200 THEN MB_MASTER.wREAD_QUANTITY:=2; ELSE
							  MB_MASTER.wREAD_QUANTITY:=VARS[VarCnt].Variable_Size;
							END_IF
							MB_MASTER.wWRITE_ADDRESS:=0;
							MB_MASTER.wWRITE_QUANTITY:=0;
					END_CASE
					VarRetry:=0;
					MB_Start:=TRUE;
				ELSE
					VarCnt:=VarCnt+1;
				END_IF
			END_WHILE
			(* Check loop completed -> no actions *)
			IF VarSta=2 THEN VarSta:=1; END_IF
		END_IF

	3: (* === Wait & process MB response *)
		IF NOT MB_Start THEN
			IF MB_MASTER.wERROR=0 THEN
				CASE VARS[VarCnt].FunCode OF
					1,2,3,4:
						IF VARS[VarCnt].Variable_Size=200 THEN
							COPY_32SWAP16(ADR(MB_READBUF), VARS[VarCnt].Variable);
						ELSIF VARS[VarCnt].Variable_Size>1 THEN
							MEMCPY(ADR(MB_READBUF), VARS[VarCnt].Variable, 2*VARS[VarCnt].Variable_Size);
						ELSE
							VARS[VarCnt].Variable^:=MB_READBUF[0];
						END_IF
				END_CASE
				MB_Lock:=FALSE;
				(* Signal error recovery *)
				IF VARS_Alarm=TRUE AND VarCnt=VarAlarm THEN
					LogEv(EL_Wrn,EO_MODBUS_TCP,ID,5,'');
					VARS_Alarm:=FALSE;
				END_IF
				(* Next var *)
				VarCnt:=VarCnt+1;
				VarSta:=2;
			ELSE
				IF VarRetry<10 THEN
					VarRetry:=VarRetry+1;
					MB_Start:=TRUE;
				ELSE
					MB_Lock:=FALSE;
					(* Signal error *)
					IF VARS_Alarm=FALSE THEN
						LogEv(EL_Wrn,EO_MODBUS_TCP,ID,3,WORD_TO_STRING(MB_MASTER.wERROR));
						VARS_Alarm:=TRUE;
						VarAlarm:=VarCnt-1;
					END_IF
					(* Next var *)
					VarCnt:=VarCnt+1;
					VarSta:=2;
				END_IF
			END_IF
		END_IF

ELSE
	VarSta:=0;
END_CASE
END_ACTION

(* POU Utils Functions/PLANT_STATUS, ST *)
FUNCTION_BLOCK PLANT_STATUS
VAR_INPUT
	obj_Status		:	WORD;
END_VAR
VAR_OUTPUT
END_VAR
VAR
	PLANT_STATUS	:	WORD;

	Pwm				:	TON := (PT:=T#1s);
END_VAR
CASE plant_Status OF

	0:	(* Plant OK - Everything works well *)
		Pwm(IN:=FALSE);							(* Stop timer if running *)
		LAMP_AL := FALSE;						(* Keep the lamp switched off *)

	1:	(* Plant in warning *)
		Pwm(IN:= NOT(Pwm.Q));

		IF Pwm.Q THEN
			LAMP_AL := NOT LAMP_AL;				(* Toggle output *)
		END_IF

	2:	(* Plant in alarm *)
		Pwm(IN:=FALSE);							(* Stop timer if running *)
		LAMP_AL	:= TRUE;						(* Keep the lamp switched on *)

END_CASE

plant_Status := 0;		(* Reset plant status *)
END_FUNCTION_BLOCK
ACTION UpdateStatus:
IF plant_Status = 2 THEN

	RETURN;					(* If plant already in alarm condition do nothing *)

ELSE

		IF obj_Status <> 0 THEN
			plant_Status := obj_Status;			(* If plant in warning/normal condition and current object in alarm, update plant status *)
		END_IF
END_IF
END_ACTION

(* POU PLC_WDT, ST *)
FUNCTION PLC_WDT: DWORD VAR_INPUT dwEvent: DWORD; dwFilter: DWORD; dwOwner: DWORD; END_VAR
LogEv(EL_AlarmStop,EO_SYS,1,10,'Watchdog');
END_FUNCTION

(* POU String/pSTRCAT, ST *)
(* STRCAT := STRCAT(STR1,STR2); *)
FUNCTION pSTRCAT : STRING(500)
VAR_INPUT
	STR1:	STRING(500);
	STR2:	STRING(32);
END_VAR
VAR
	ps1: POINTER TO BYTE;
	ps2: POINTER TO BYTE;
	pf:	 POINTER TO BYTE;

	ii: WORD;

END_VAR

(* versione sostitutiva thread safe della funzione CONCAT *)
(* questa funzione nasce dall'esigenza di non usare la funzione di sistema STRCAT perchè non è task safe *)

ps1 := ADR(STR1);
ps2 := ADR(STR2);

pf	:= ADR(pSTRCAT);

ii := 0;
WHILE ps1^<>0 DO
	pf^ := ps1^;
	pf := pf + 1;
	ps1:= ps1 + 1;
	ii := ii + 1;
	IF ii> 1000 THEN
		EXIT; (* termina ciclo se dimensione stringa 1 eccede per qualche motivo *)
	END_IF;

END_WHILE


WHILE ps2^<>0 DO
	pf^ := ps2^;
	pf := pf + 1;
	ps2:= ps2 + 1;
	ii := ii + 1;
	IF ii> 1000 THEN
		EXIT; (* termina ciclo se dimensione stringa 1 eccede per qualche motivo *)
	END_IF;
END_WHILE

pf^ := 0; (* termino stringa *)
END_FUNCTION

(* POU RAWTOHEXSTR, ST *)
FUNCTION RAWTOHEXSTR : STRING(128)
VAR_INPUT
	pData: POINTER TO BYTE;
	DataLen: BYTE;
END_VAR
VAR
	pt: POINTER TO BYTE;
	xl: BYTE;
END_VAR
pt:=ADR(RAWTOHEXSTR);

xl:=2;

WHILE DataLen>0 AND xl<128 DO

	pt^ := (pData^ / 16#10) + 48 + (((pData^ / 16#10)/10)*7);
	pt:=pt+1;
	pt^ := (pData^ AND 16#0F)  + 48 + (((pData^ AND 16#0F)/10)*7);
	pt:=pt+1;

	xl:=xl+2;

	DataLen:=DataLen-1;
	pData:=pData+1;

END_WHILE

pt^:=0;
END_FUNCTION

(* POU Utils/RTC_Update, ST *)
FUNCTION RTC_Update : BOOL
VAR
	T: DT;
	TS: STRING;
	TS2: STRING;
	Hour: BYTE;
	Minute: BYTE;
END_VAR
(* Get RTC time *)
T:=SysRtcGetTime(TRUE);
Sys.Time_CT_DT:=T;
(* Calculate variables *)
TS:=DT_TO_STRING(T);
Sys.Time_LogString:=DELETE(STR:=TS, LEN:=3, POS:=1);
TS2:=MID(STR:=TS, LEN:=4, POS:= 4); Sys.Time_Year 	:=STRING_TO_WORD(TS2);
TS2:=MID(STR:=TS, LEN:=2, POS:= 9); Sys.Time_Month	:=STRING_TO_BYTE(TS2);
TS2:=MID(STR:=TS, LEN:=2, POS:=12); Sys.Time_Day  	:=STRING_TO_BYTE(TS2);
Sys.Time_CT_Day:=(32*(Sys.Time_Month-1)+Sys.Time_Day-1);
TS2:=MID(STR:=TS, LEN:=2, POS:=15); Hour			:=STRING_TO_BYTE(TS2);
TS2:=MID(STR:=TS, LEN:=2, POS:=18); Minute		 	:=STRING_TO_BYTE(TS2);
Sys.Time_CT_Quarter:=Hour*4+(Minute/15);
END_FUNCTION

(* POU Utils Functions/SHIFT_ARRAY, ST *)
FUNCTION SHIFT_ARRAY : BOOL
VAR_INPUT
	pData	:	POINTER TO ARRAY [1..2] OF WORD;
	Size	:	BYTE;
END_VAR
VAR
	pNew	:	POINTER TO WORD;
	i		:	BYTE;
END_VAR
(* Shift right *)
FOR i:=1 TO (Size-1) BY 1 DO

	(*pNew := pData + 1;*)
	pData^[i] := pData^[i+1];
	(*pData := pData + 1;*)

END_FOR
END_FUNCTION

(* Visualisation PLC_VIS_CicloAUTO
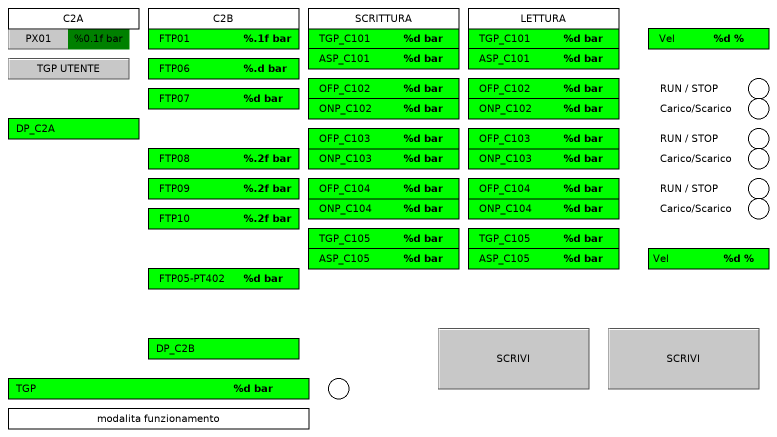
rectangle at (170,350)-(321,371): text "DP_C2B"
rectangle at (330,210)-(481,231): text "ONP_C104"
rectangle at (330,190)-(481,211): text "OFP_C104"
rectangle at (330,160)-(481,181): text "ONP_C103"
rectangle at (330,140)-(481,161): text "OFP_C103"
button at (30,40)-(91,61): text "PX01"
rectangle at (90,40)-(151,61): text "%0.1f bar"; shows INT_TO_REAL(.PX01.ValoreScalato)/10
rectangle at (170,40)-(321,61): text "FTP01"
rectangle at (260,40)-(321,61): text "%.1f bar"; shows .FPT01.PressioneCalcolata
rectangle at (170,70)-(321,91): text "FTP06"
rectangle at (170,100)-(321,121): text "FTP07"
rectangle at (170,160)-(321,181): text "FTP08"
rectangle at (170,190)-(321,211): text "FTP09"
rectangle at (170,220)-(321,241): text "FTP10"
rectangle at (330,40)-(481,61): text "TGP_C101"
rectangle at (420,40)-(481,61): text "%d bar"; shows PLC_PRG.TGP_C101
rectangle at (330,60)-(481,81): text "ASP_C101"
rectangle at (420,60)-(481,81): text "%d bar"; shows PLC_PRG.ASP_C101
rectangle at (330,90)-(481,111): text "OFP_C102"
rectangle at (420,90)-(481,111): text "%d bar"; shows PLC_PRG.OFP_C102
rectangle at (330,110)-(481,131): text "ONP_C102"
rectangle at (420,110)-(481,131): text "%d bar"; shows PLC_PRG.ONP_C102
rectangle at (420,140)-(481,161): text "%d bar"; shows PLC_PRG.OFP_C103
rectangle at (420,160)-(481,181): text "%d bar"; shows PLC_PRG.ONP_C103
rectangle at (420,190)-(481,211): text "%d bar"; shows PLC_PRG.OFP_C104
rectangle at (420,210)-(481,231): text "%d bar"; shows PLC_PRG.ONP_C104
rectangle at (330,240)-(481,261): text "TGP_C105"
rectangle at (420,240)-(481,261): text "%d bar"; shows PLC_PRG.TGP_C105
rectangle at (330,260)-(481,281): text "ASP_C105"
rectangle at (420,260)-(481,281): text "%d bar"; shows PLC_PRG.ASP_C105
rectangle at (490,210)-(641,231): text "ONP_C104"
rectangle at (490,190)-(641,211): text "OFP_C104"
rectangle at (490,160)-(641,181): text "ONP_C103"
rectangle at (490,140)-(641,161): text "OFP_C103"
rectangle at (490,40)-(641,61): text "TGP_C101"
rectangle at (580,40)-(641,61): text "%d bar"; shows .COMPRESSORE01.MB_RegistriHoldingLetti[112]
rectangle at (490,60)-(641,81): text "ASP_C101"
rectangle at (580,60)-(641,81): text "%d bar"; shows .COMPRESSORE01.MB_RegistriHoldingLetti[113]
rectangle at (490,90)-(641,111): text "OFP_C102"
rectangle at (580,90)-(641,111): text "%d bar"; shows .COMPRESSORE02.MB_RegistriHoldingLetti[112]
rectangle at (490,110)-(641,131): text "ONP_C102"
rectangle at (580,110)-(641,131): text "%d bar"; shows .COMPRESSORE02.MB_RegistriHoldingLetti[113]
rectangle at (580,140)-(641,161): text "%d bar"; shows .COMPRESSORE03.MB_RegistriHoldingLetti[112]
rectangle at (580,160)-(641,181): text "%d bar"; shows .COMPRESSORE03.MB_RegistriHoldingLetti[113]
rectangle at (580,190)-(641,211): text "%d bar"; shows .COMPRESSORE04.MB_RegistriHoldingLetti[112]
rectangle at (580,210)-(641,231): text "%d bar"; shows .COMPRESSORE04.MB_RegistriHoldingLetti[113]
rectangle at (490,240)-(641,261): text "TGP_C105"
rectangle at (580,240)-(641,261): text "%d bar"; shows .COMPRESSORE05.MB_RegistriHoldingLetti[112]
rectangle at (490,260)-(641,281): text "ASP_C105"
rectangle at (580,260)-(641,281): text "%d bar"; shows .COMPRESSORE05.MB_RegistriHoldingLetti[113]
rectangle at (170,280)-(321,301): text "FTP05-PT402"
rectangle at (260,280)-(321,301): text "%d bar"; shows .FPT05.Parametro32
rectangle at (30,390)-(331,411): text "TGP"
rectangle at (250,390)-(311,411): text "%d bar"; shows PLC_PRG.TGP
rectangle at (670,40)-(791,61): text "Vel"
rectangle at (730,40)-(791,61): text "%d %"; shows .COMPRESSORE01.MB_RegistriHoldingLetti[20]
rectangle at (670,260)-(791,281): text "Vel"
rectangle at (740,260)-(791,281): text "%d %"; shows .COMPRESSORE05.MB_RegistriHoldingLetti[20]
ellipse at (770,90)-(791,111): alarm colour if .COMPRESSORE02.StatusControl[1]
ellipse at (770,110)-(791,131): alarm colour if .COMPRESSORE02.StatusControl[2]
rectangle at (680,90)-(771,111): text "RUN / STOP"
rectangle at (680,110)-(771,131): text "Carico/Scarico"
ellipse at (770,140)-(791,161): alarm colour if .COMPRESSORE03.StatusControl[1]
ellipse at (770,160)-(791,181): alarm colour if .COMPRESSORE03.StatusControl[2]
rectangle at (680,140)-(771,161): text "RUN / STOP"
rectangle at (680,160)-(771,181): text "Carico/Scarico"
ellipse at (770,190)-(791,211): alarm colour if .COMPRESSORE04.StatusControl[1]
ellipse at (770,210)-(791,231): alarm colour if .COMPRESSORE04.StatusControl[2]
rectangle at (680,190)-(771,211): text "RUN / STOP"
rectangle at (680,210)-(771,231): text "Carico/Scarico"
button at (30,70)-(151,91): text "TGP UTENTE"
rectangle at (330,20)-(481,41): text "SCRITTURA"
rectangle at (490,20)-(641,41): text "LETTURA"
rectangle at (260,220)-(321,241): text "%.2f bar"; shows .FPT10.IntPressioneCalcolata
rectangle at (260,190)-(321,211): text "%.2f bar"; shows .FPT09.IntPressioneCalcolata
rectangle at (260,160)-(321,181): text "%.2f bar"; shows .FPT08.IntPressioneCalcolata
rectangle at (260,100)-(321,121): text "%d bar"; shows .FPT07.Parametro32
rectangle at (260,70)-(321,91): text "%.d bar"; shows .FPT06.IntPressioneCalcolata
rectangle at (170,20)-(321,41): text "C2B"
rectangle at (30,20)-(161,41): text "C2A"
rectangle at (30,130)-(161,151): text "DP_C2A"
button at (630,340)-(781,401): text "SCRIVI"; toggles PLC_PRG.HMISTART
rectangle at (30,420)-(331,441): text "modalita funzionamento"
button at (460,340)-(611,401): text "SCRIVI"; toggles PLC_PRG.HMISTART03
ellipse at (350,390)-(371,411): alarm colour if PLC_PRG.Ton_pausaTrig.Q
6 elements of other kinds (tables, trends, ...) not read
*)

(* Visualisation PLC_VISU
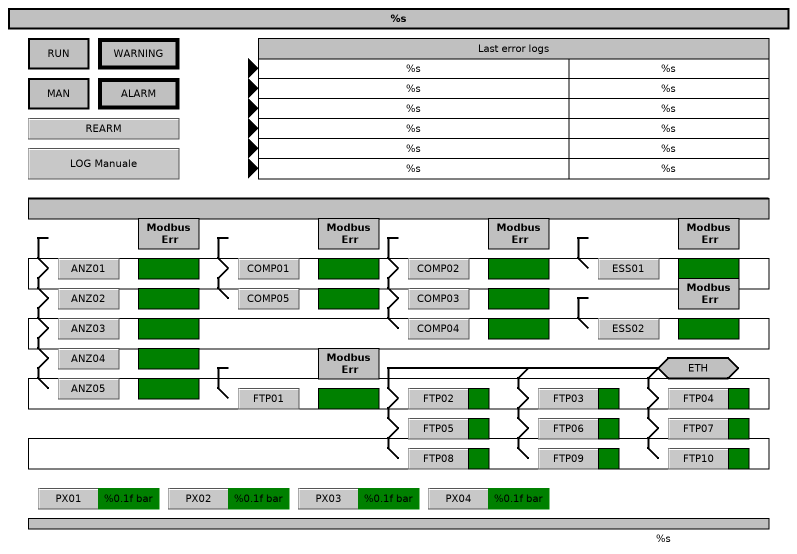
rectangle at (10,0)-(791,21): text "%s"; shows .Plant_NAME
rounded rectangle at (30,30)-(91,61): text "RUN"; alarm colour if NOT Mode_Manual; runs INTERN ASSIGN Mode_Manual:=(FALSE)
rounded rectangle at (30,70)-(91,101): text "MAN"; alarm colour if Mode_Manual; runs INTERN ASSIGN Mode_Manual:=(TRUE)
rectangle at (570,50)-(771,71): text "%s"; shows Sys.LastLogs_Msg[0]
polygon at (250,150)-(260,170): invisible if Sys.LastLogs_Idx<>0
rectangle at (570,70)-(771,91): text "%s"; shows Sys.LastLogs_Msg[1]
polygon at (250,50)-(260,70): invisible if Sys.LastLogs_Idx<>1
rectangle at (570,90)-(771,111): text "%s"; shows Sys.LastLogs_Msg[2]
polygon at (250,70)-(260,90): invisible if Sys.LastLogs_Idx<>2
rectangle at (570,110)-(771,131): text "%s"; shows Sys.LastLogs_Msg[3]
polygon at (250,90)-(260,110): invisible if Sys.LastLogs_Idx<>3
rectangle at (570,130)-(771,151): text "%s"; shows Sys.LastLogs_Msg[4]
polygon at (250,110)-(260,130): invisible if Sys.LastLogs_Idx<>4
rectangle at (570,150)-(771,171): text "%s"; shows Sys.LastLogs_Msg[5]
polygon at (250,130)-(260,150): invisible if Sys.LastLogs_Idx<>5
rectangle at (260,50)-(571,71): text "%s"; shows Sys.LastLogs_Dat[0]
rectangle at (260,70)-(571,91): text "%s"; shows Sys.LastLogs_Dat[1]
rectangle at (260,90)-(571,111): text "%s"; shows Sys.LastLogs_Dat[2]
rectangle at (260,110)-(571,131): text "%s"; shows Sys.LastLogs_Dat[3]
rectangle at (260,130)-(571,151): text "%s"; shows Sys.LastLogs_Dat[4]
rectangle at (260,150)-(571,171): text "%s"; shows Sys.LastLogs_Dat[5]
rectangle at (100,70)-(181,101): text "ALARM"; alarm colour if Sys.Alarm; runs INTERN ASSIGN Mode_Manual:=(FALSE)
rectangle at (100,30)-(181,61): text "WARNING"; alarm colour if Sys.Warning; runs INTERN ASSIGN Mode_Manual:=(TRUE)
button at (30,110)-(181,131): text "REARM"; runs INTERN ASSIGN Sys.Alarm:=(FALSE);INTERN ASSIGN Sys.Warning:=(FALSE)
button at (60,250)-(121,271): text "ANZ01"
rectangle at (260,30)-(771,51): text "Last error logs"
button at (60,280)-(121,301): text "ANZ02"
rectangle at (560,520)-(771,541): text "%s"; shows Sys.Time_LogString
rectangle at (140,210)-(201,241): text "Modbus / Err"
rectangle at (140,280)-(201,301): alarm colour if ANZ_MODBUS_CONNECTOR_INEPRO[2].fTimeout
button at (60,310)-(121,331): text "ANZ03"
rectangle at (140,310)-(201,331): alarm colour if ANZ_MODBUS_CONNECTOR_INEPRO[3].fTimeout
rectangle at (140,250)-(201,271): alarm colour if ANZ_MODBUS_CONNECTOR_INEPRO[1].fTimeout
button at (60,340)-(121,361): text "ANZ04"
rectangle at (140,340)-(201,361): alarm colour if ANZ_MODBUS_CONNECTOR_INEPRO[4].fTimeout
button at (60,370)-(121,391): text "ANZ05"
rectangle at (140,370)-(201,391): alarm colour if ANZ_MODBUS_CONNECTOR_INEPRO[5].fTimeout
button at (240,250)-(301,271): text "COMP01"
button at (240,280)-(301,301): text "COMP05"
rectangle at (320,250)-(381,271): alarm colour if .COMPRESSORE01.ErroreComuModBus
rectangle at (320,280)-(381,301): alarm colour if .COMPRESSORE05.ErroreComuModBus
rectangle at (320,210)-(381,241): text "Modbus / Err"
button at (410,250)-(471,271): text "COMP02"
button at (410,280)-(471,301): text "COMP03"
rectangle at (490,250)-(551,271): alarm colour if .COMPRESSORE02.ErroreComuModBus
rectangle at (490,280)-(551,301): alarm colour if .COMPRESSORE03.ErroreComuModBus
rectangle at (490,210)-(551,241): text "Modbus / Err"
button at (600,250)-(661,271): text "ESS01"
button at (600,310)-(661,331): text "ESS02"
rectangle at (680,250)-(741,271): alarm colour if ESSICATORE01.ErroreComuModBus
rectangle at (680,310)-(741,331): alarm colour if ESSICATORE02.ErroreComuModBus
rectangle at (680,210)-(741,241): text "Modbus / Err"
button at (240,380)-(301,401): text "FTP01"
rectangle at (320,380)-(381,401): alarm colour if .FPT01.ErroreComuModBus
rectangle at (320,340)-(381,371): text "Modbus / Err"
button at (410,310)-(471,331): text "COMP04"
rectangle at (490,310)-(551,331): alarm colour if .COMPRESSORE04.ErroreComuModBus
button at (40,480)-(101,501): text "PX01"
rectangle at (100,480)-(161,501): text "%0.1f bar"; shows INT_TO_REAL(.PX01.ValoreScalato)/10
button at (170,480)-(231,501): text "PX02"
rectangle at (230,480)-(291,501): text "%0.1f bar"; shows INT_TO_REAL(.PX02.ValoreScalato)/10
button at (300,480)-(361,501): text "PX03"
rectangle at (360,480)-(421,501): text "%0.1f bar"; shows INT_TO_REAL(.PX03.ValoreScalato)/10
button at (430,480)-(491,501): text "PX04"
rectangle at (490,480)-(551,501): text "%0.1f bar"; shows INT_TO_REAL(.PX04.ValoreScalato)/10
button at (30,140)-(181,171): text "LOG Manuale"; taps PLC_PRG.HMI_AggiornaLog
button at (410,380)-(471,401): text "FTP02"
polygon at (660,350)-(740,370): text "ETH"
rectangle at (470,380)-(491,401): alarm colour if .FPT02.ErroreComuModBus
button at (540,380)-(601,401): text "FTP03"
rectangle at (600,380)-(621,401): alarm colour if .FPT03.ErroreComuModBus
button at (670,380)-(731,401): text "FTP04"
rectangle at (730,380)-(751,401): alarm colour if .FPT04.ErroreComuModBus
button at (410,410)-(471,431): text "FTP05"
rectangle at (470,410)-(491,431): alarm colour if .FPT05.ErroreComuModBus
button at (540,410)-(601,431): text "FTP06"
rectangle at (600,410)-(621,431): alarm colour if .FPT06.ErroreComuModBus
button at (670,410)-(731,431): text "FTP07"
rectangle at (730,410)-(751,431): alarm colour if .FPT07.ErroreComuModBus
button at (670,440)-(731,461): text "FTP10"
rectangle at (730,440)-(751,461): alarm colour if .FPT10.ErroreComuModBus
button at (540,440)-(601,461): text "FTP09"
rectangle at (600,440)-(621,461): alarm colour if .FPT09.ErroreComuModBus
button at (410,440)-(471,461): text "FTP08"
rectangle at (470,440)-(491,461): alarm colour if .FPT08.ErroreComuModBus
rectangle at (680,270)-(741,301): text "Modbus / Err"
29 more shapes without text or variables
28 elements of other kinds (tables, trends, ...) not read
*)

